LIN {X 0,Y 291.702,Z 865.941,A -85,B 0,C 180,E1 -16752.169,E2 -16752.169} C_VEL
LIN {X 0,Y 292.746,Z 856.676,A -85,B 0,C 180,E1 -16754.244,E2 -16754.244} C_VEL
LIN {X 0,Y 293.945,Z 846.153,A -85,B 0,C 180,E1 -16756.136,E2 -16756.136} C_VEL
LIN {X 0,Y 295.045,Z 835.726,A -85,B 0,C 180,E1 -16757.673,E2 -16757.673} C_VEL
LIN {X 0,Y 296.142,Z 824.245,A -85,B 0,C 180,E1 -16759.044,E2 -16759.044} C_VEL
LIN {X 0,Y 296.402,Z 819.576,A -85,B 0,C 180,E1 -16759.528,E2 -16759.528} C_VEL
LIN {X 0,Y 293.776,Z 806.153,A -85,B 0,C 180,E1 -16760.832,E2 -16760.832} C_VEL
LIN {X 0,Y 290.876,Z 792.284,A -85,B 0,C 180,E1 -16761.882,E2 -16761.882} C_VEL
LIN {X 0,Y 290.051,Z 788.06,A -85,B 0,C 180,E1 -16762.151,E2 -16762.151} C_VEL
LIN {X 0,Y 290.084,Z 786.203,A -85,B 0,C 180,E1 -16764.32,E2 -16764.32} C_VEL
LIN {X 0,Y 290.234,Z 785.335,A -85,B 0,C 180,E1 -16765.839,E2 -16765.839} C_VEL
LIN {X 0,Y 290.606,Z 785.282,A -85,B 0,C 180,E1 -16769.469,E2 -16769.469} C_VEL
LIN {X 0,Y 290.945,Z 785.244,A -85,B 0,C 180,E1 -16772.279,E2 -16772.279} C_VEL
LIN {X 0,Y 291.204,Z 785.208,A -85,B 0,C 180,E1 -16775.394,E2 -16775.394} C_VEL
LIN {X 0,Y 291.336,Z 785.194,A -85,B 0,C 180,E1 -16778.842,E2 -16778.842} C_VEL
LIN {X 0,Y 291.315,Z 785.197,A -85,B 0,C 180,E1 -16782.491,E2 -16782.491} C_VEL
LIN {X 0,Y 291.303,Z 785.198,A -85,B 0,C 180,E1 -16786.365,E2 -16786.365} C_VEL
LIN {X 0,Y 291.372,Z 785.188,A -85,B 0,C 180,E1 -16790.518,E2 -16790.518} C_VEL
LIN {X 0,Y 291.398,Z 785.189,A -85,B 0,C 180,E1 -16792.918,E2 -16792.918} C_VEL
LIN {X 0,Y 291.337,Z 785.192,A -85,B 0,C 180,E1 -16796.3,E2 -16796.3} C_VEL
LIN {X 0,Y 291.358,Z 785.188,A -85,B 0,C 180,E1 -16800.267,E2 -16800.267} C_VEL
LIN {X 0,Y 291.351,Z 785.19,A -85,B 0,C 180,E1 -16804.266,E2 -16804.266} C_VEL
LIN {X 0,Y 291.361,Z 785.193,A -85,B 0,C 180,E1 -16807.298,E2 -16807.298} C_VEL
LIN {X 0,Y 291.398,Z 785.184,A -85,B 0,C 180,E1 -16810.266,E2 -16810.266} C_VEL
LIN {X 0,Y 291.489,Z 785.172,A -85,B 0,C 180,E1 -16814.665,E2 -16814.665} C_VEL
LIN {X 0,Y 291.52,Z 785.169,A -85,B 0,C 180,E1 -16818.88,E2 -16818.88} C_VEL
LIN {X 0,Y 291.642,Z 785.158,A -85,B 0,C 180,E1 -16821.687,E2 -16821.687} C_VEL
LIN {X 0,Y 291.586,Z 785.16,A -85,B 0,C 180,E1 -16824.467,E2 -16824.467} C_VEL
LIN {X 0,Y 291.86,Z 785.127,A -85,B 0,C 180,E1 -16828.62,E2 -16828.62} C_VEL
LIN {X 0,Y 291.859,Z 785.127,A -85,B 0,C 180,E1 -16831.38,E2 -16831.38} C_VEL
LIN {X 0,Y 291.676,Z 785.15,A -85,B 0,C 180,E1 -16836.92,E2 -16836.92} C_VEL
LIN {X 0,Y 291.558,Z 785.165,A -85,B 0,C 180,E1 -16839.714,E2 -16839.714} C_VEL
LIN {X 0,Y 291.506,Z 785.171,A -85,B 0,C 180,E1 -16843.951,E2 -16843.951} C_VEL
LIN {X 0,Y 291.42,Z 785.184,A -85,B 0,C 180,E1 -16846.822,E2 -16846.822} C_VEL
LIN {X 0,Y 291.416,Z 785.182,A -85,B 0,C 180,E1 -16849.861,E2 -16849.861} C_VEL
LIN {X 0,Y 291.352,Z 785.191,A -85,B 0,C 180,E1 -16854.21,E2 -16854.21} C_VEL
LIN {X 0,Y 291.346,Z 785.192,A -85,B 0,C 180,E1 -16857.279,E2 -16857.279} C_VEL
LIN {X 0,Y 291.311,Z 785.196,A -85,B 0,C 180,E1 -16860.44,E2 -16860.44} C_VEL
LIN {X 0,Y 291.337,Z 785.192,A -85,B 0,C 180,E1 -16863.7,E2 -16863.7} C_VEL
LIN {X 0,Y 291.366,Z 785.191,A -85,B 0,C 180,E1 -16867.254,E2 -16867.254} C_VEL
LIN {X 0,Y 291.327,Z 785.193,A -85,B 0,C 180,E1 -16870.644,E2 -16870.644} C_VEL
LIN {X 0,Y 291.284,Z 785.198,A -85,B 0,C 180,E1 -16874.403,E2 -16874.403} C_VEL
LIN {X 0,Y 291.321,Z 785.193,A -85,B 0,C 180,E1 -16878.406,E2 -16878.406} C_VEL
LIN {X 0,Y 291.337,Z 785.194,A -85,B 0,C 180,E1 -16881.158,E2 -16881.158} C_VEL
LIN {X 0,Y 291.364,Z 785.189,A -85,B 0,C 180,E1 -16882.915,E2 -16882.915} C_VEL
LIN {X 0,Y 291.12,Z 785.219,A -85,B 0,C 180,E1 -16886.274,E2 -16886.274} C_VEL
LIN {X 0,Y 290.791,Z 785.263,A -85,B 0,C 180,E1 -16889.502,E2 -16889.502} C_VEL
LIN {X 0,Y 290.405,Z 785.308,A -85,B 0,C 180,E1 -16892.627,E2 -16892.627} C_VEL
LIN {X 0,Y 289.99,Z 785.385,A -85,B 0,C 180,E1 -16896.052,E2 -16896.052} C_VEL
LIN {X 0,Y 290.009,Z 787.302,A -85,B 0,C 180,E1 -16898.005,E2 -16898.005} C_VEL
LIN {X 0,Y 292.931,Z 801.867,A -85,B 0,C 180,E1 -16899.012,E2 -16899.012} C_VEL
LIN {X 0,Y 295.424,Z 814.684,A -85,B 0,C 180,E1 -16900.163,E2 -16900.163} C_VEL
LIN {X 0,Y 296.257,Z 818.937,A -85,B 0,C 180,E1 -16900.604,E2 -16900.604} C_VEL
LIN {X 0,Y 295.466,Z 830.012,A -85,B 0,C 180,E1 -16901.81,E2 -16901.81} C_VEL
LIN {X 0,Y 294.374,Z 841.527,A -85,B 0,C 180,E1 -16903.354,E2 -16903.354} C_VEL
LIN {X 0,Y 293.182,Z 851.897,A -85,B 0,C 180,E1 -16905.068,E2 -16905.068} C_VEL
LIN {X 0,Y 292.179,Z 860.521,A -85,B 0,C 180,E1 -16906.792,E2 -16906.792} C_VEL
LIN {X 0,Y 291.27,Z 869.021,A -85,B 0,C 180,E1 -16908.872,E2 -16908.872} C_VEL
LIN {X 0,Y 290.529,Z 875.88,A -85,B 0,C 180,E1 -16910.955,E2 -16910.955} C_VEL
LIN {X 0,Y 290.145,Z 881.419,A -85,B 0,C 180,E1 -16913.045,E2 -16913.045} C_VEL
LIN {X 0,Y 289.874,Z 885.775,A -85,B 0,C 180,E1 -16915.134,E2 -16915.134} C_VEL
LIN {X 0,Y 289.725,Z 889.058,A -85,B 0,C 180,E1 -16917.221,E2 -16917.221} C_VEL
LIN {X 0,Y 289.68,Z 890.166,A -85,B 0,C 180,E1 -16918.16,E2 -16918.16} C_VEL
LIN {X 0,Y 289.052,Z 891.419,A -85,B 0,C 180,E1 -16919.297,E2 -16919.297} C_VEL
LIN {X 0,Y 286.375,Z 892.977,A -85,B 0,C 180,E1 -16921.173,E2 -16921.173} C_VEL
LIN {X 0,Y 284.14,Z 893.629,A -85,B 0,C 180,E1 -16922.707,E2 -16922.707} C_VEL
LIN {X 0,Y 283.223,Z 893.7,A -85,B 0,C 180,E1 -16923.895,E2 -16923.895} C_VEL
LIN {X 0,Y 283.171,Z 893.633,A -85,B 0,C 180,E1 -16924.296,E2 -16924.296} C_VEL
LIN {X 0,Y 283.733,Z 892.595,A -85,B 0,C 180,E1 -16927.116,E2 -16927.116} C_VEL
LIN {X 0,Y 284.867,Z 890.681,A -85,B 0,C 180,E1 -16929.301,E2 -16929.301} C_VEL
LIN {X 0,Y 286.349,Z 886.93,A -85,B 0,C 180,E1 -16932.043,E2 -16932.043} C_VEL
LIN {X 0,Y 288.523,Z 881.299,A -85,B 0,C 180,E1 -16934.82,E2 -16934.82} C_VEL
LIN {X 0,Y 290.974,Z 874.766,A -85,B 0,C 180,E1 -16937.212,E2 -16937.212} C_VEL
LIN {X 0,Y 293.868,Z 866.526,A -85,B 0,C 180,E1 -16939.563,E2 -16939.563} C_VEL
LIN {X 0,Y 296.798,Z 857.782,A -85,B 0,C 180,E1 -16941.534,E2 -16941.534} C_VEL
LIN {X 0,Y 300.013,Z 847.159,A -85,B 0,C 180,E1 -16943.469,E2 -16943.469} C_VEL
LIN {X 0,Y 302.761,Z 837.452,A -85,B 0,C 180,E1 -16944.894,E2 -16944.894} C_VEL
LIN {X 0,Y 301.396,Z 829.053,A -85,B 0,C 180,E1 -16946.69,E2 -16946.69} C_VEL
LIN {X 0,Y 299.193,Z 821.542,A -85,B 0,C 180,E1 -16948.479,E2 -16948.479} C_VEL
LIN {X 0,Y 296.103,Z 814.055,A -85,B 0,C 180,E1 -16950.547,E2 -16950.547} C_VEL
LIN {X 0,Y 292.669,Z 807.234,A -85,B 0,C 180,E1 -16952.81,E2 -16952.81} C_VEL
LIN {X 0,Y 290.172,Z 802.954,A -85,B 0,C 180,E1 -16954.564,E2 -16954.564} C_VEL
LIN {X 0,Y 287.786,Z 800.116,A -85,B 0,C 180,E1 -16956.303,E2 -16956.303} C_VEL
LIN {X 0,Y 287.055,Z 798.413,A -85,B 0,C 180,E1 -16957.188,E2 -16957.188} C_VEL
LIN {X 0,Y 287.219,Z 798.097,A -85,B 0,C 180,E1 -16960.664,E2 -16960.664} C_VEL
LIN {X 0,Y 287.395,Z 798.308,A -85,B 0,C 180,E1 -16963.215,E2 -16963.215} C_VEL
LIN {X 0,Y 287.484,Z 798.802,A -85,B 0,C 180,E1 -16965.151,E2 -16965.151} C_VEL
LIN {X 0,Y 287.572,Z 799.696,A -85,B 0,C 180,E1 -16967.155,E2 -16967.155} C_VEL
LIN {X 0,Y 287.764,Z 802.16,A -85,B 0,C 180,E1 -16970.58,E2 -16970.58} C_VEL
LIN {X 0,Y 287.97,Z 805.028,A -85,B 0,C 180,E1 -16973.185,E2 -16973.185} C_VEL
LIN {X 0,Y 290.424,Z 811.895,A -85,B 0,C 180,E1 -16975.365,E2 -16975.365} C_VEL
LIN {X 0,Y 292.114,Z 817.637,A -85,B 0,C 180,E1 -16976.764,E2 -16976.764} C_VEL
LIN {X 0,Y 293.714,Z 824.775,A -85,B 0,C 180,E1 -16978.236,E2 -16978.236} C_VEL
LIN {X 0,Y 295.55,Z 834.314,A -85,B 0,C 180,E1 -16980.042,E2 -16980.042} C_VEL
LIN {X 0,Y 296.936,Z 846.854,A -85,B 0,C 180,E1 -16982.195,E2 -16982.195} C_VEL
LIN {X 0,Y 297.261,Z 857.519,A -85,B 0,C 180,E1 -16983.953,E2 -16983.953} C_VEL
LIN {X 0,Y 296.48,Z 867.317,A -85,B 0,C 180,E1 -16985.542,E2 -16985.542} C_VEL
LIN {X 0,Y 295.029,Z 876.946,A -85,B 0,C 180,E1 -16987.226,E2 -16987.226} C_VEL
LIN {X 0,Y 291.992,Z 887.534,A -85,B 0,C 180,E1 -16989.205,E2 -16989.205} C_VEL
LIN {X 0,Y 289.317,Z 896.401,A -85,B 0,C 180,E1 -16991.261,E2 -16991.261} C_VEL
LIN {X 0,Y 287.218,Z 903.602,A -85,B 0,C 180,E1 -16993.291,E2 -16993.291} C_VEL
LIN {X 0,Y 285.274,Z 910.592,A -85,B 0,C 180,E1 -16995.738,E2 -16995.738} C_VEL
LIN {X 0,Y 284.001,Z 915.383,A -85,B 0,C 180,E1 -16997.857,E2 -16997.857} C_VEL
LIN {X 0,Y 283.201,Z 919.135,A -85,B 0,C 180,E1 -16999.996,E2 -16999.996} C_VEL
LIN {X 0,Y 282.607,Z 922.647,A -85,B 0,C 180,E1 -17002.857,E2 -17002.857} C_VEL
LIN {X 0,Y 282.567,Z 923.809,A -85,B 0,C 180,E1 -17004.29,E2 -17004.29} C_VEL
LIN {X 0,Y 282.529,Z 924.564,A -85,B 0,C 180,E1 -17005.72,E2 -17005.72} C_VEL
LIN {X 0,Y 282.847,Z 924.892,A -85,B 0,C 180,E1 -17008.576,E2 -17008.576} C_VEL
LIN {X 0,Y 282.886,Z 925.833,A -85,B 0,C 180,E1 -17010,E2 -17010} C_VEL
LIN {X 0,Y 282.634,Z 926.326,A -85,B 0,C 180,E1 -17011.425,E2 -17011.425} C_VEL
LIN {X 0,Y 282.506,Z 926.418,A -85,B 0,C 180,E1 -17012.852,E2 -17012.852} C_VEL
LIN {X 0,Y 282.491,Z 926.109,A -85,B 0,C 180,E1 -17014.28,E2 -17014.28} C_VEL
LIN {X 0,Y 282.487,Z 925.361,A -85,B 0,C 180,E1 -17015.711,E2 -17015.711} C_VEL
LIN {X 0,Y 282.82,Z 922.66,A -85,B 0,C 180,E1 -17018.575,E2 -17018.575} C_VEL
LIN {X 0,Y 283.413,Z 919.571,A -85,B 0,C 180,E1 -17020.719,E2 -17020.719} C_VEL
LIN {X 0,Y 284.314,Z 915.533,A -85,B 0,C 180,E1 -17022.854,E2 -17022.854} C_VEL
LIN {X 0,Y 285.869,Z 910.437,A -85,B 0,C 180,E1 -17024.96,E2 -17024.96} C_VEL
LIN {X 0,Y 287.926,Z 903.011,A -85,B 0,C 180,E1 -17027.445,E2 -17027.445} C_VEL
LIN {X 0,Y 290.527,Z 894.081,A -85,B 0,C 180,E1 -17029.796,E2 -17029.796} C_VEL
LIN {X 0,Y 293.508,Z 884.684,A -85,B 0,C 180,E1 -17031.786,E2 -17031.786} C_VEL
LIN {X 0,Y 295.658,Z 877.383,A -85,B 0,C 180,E1 -17033.093,E2 -17033.093} C_VEL
LIN {X 0,Y 297.65,Z 865.19,A -85,B 0,C 180,E1 -17035.151,E2 -17035.151} C_VEL
LIN {X 0,Y 297.917,Z 856.285,A -85,B 0,C 180,E1 -17036.63,E2 -17036.63} C_VEL
LIN {X 0,Y 297.073,Z 845.544,A -85,B 0,C 180,E1 -17038.505,E2 -17038.505} C_VEL
LIN {X 0,Y 295.39,Z 836.08,A -85,B 0,C 180,E1 -17040.302,E2 -17040.302} C_VEL
LIN {X 0,Y 294.81,Z 833.066,A -85,B 0,C 180,E1 -17040.882,E2 -17040.882} C_VEL
LIN {X 0,Y 292.262,Z 823.462,A -85,B 0,C 180,E1 -17043.018,E2 -17043.018} C_VEL
LIN {X 0,Y 290.605,Z 818.78,A -85,B 0,C 180,E1 -17044.283,E2 -17044.283} C_VEL
LIN {X 0,Y 290.319,Z 817.311,A -85,B 0,C 180,E1 -17044.605,E2 -17044.605} C_VEL
LIN {X 0,Y 288.762,Z 814.222,A -85,B 0,C 180,E1 -17045.741,E2 -17045.741} C_VEL
LIN {X 0,Y 287.814,Z 810.336,A -85,B 0,C 180,E1 -17046.863,E2 -17046.863} C_VEL
LIN {X 0,Y 287.991,Z 808.098,A -85,B 0,C 180,E1 -17049.383,E2 -17049.383} C_VEL
LIN {X 0,Y 287.921,Z 806.691,A -85,B 0,C 180,E1 -17051.228,E2 -17051.228} C_VEL
LIN {X 0,Y 287.538,Z 804.324,A -85,B 0,C 180,E1 -17055.139,E2 -17055.139} C_VEL
LIN {X 0,Y 287.216,Z 802.831,A -85,B 0,C 180,E1 -17058.647,E2 -17058.647} C_VEL
LIN {X 0,Y 286.958,Z 801.877,A -85,B 0,C 180,E1 -17062.244,E2 -17062.244} C_VEL
LIN {X 0,Y 286.873,Z 801.861,A -85,B 0,C 180,E1 -17062.894,E2 -17062.894} C_VEL
LIN {X 0,Y 288.086,Z 804.443,A -85,B 0,C 180,E1 -17064.161,E2 -17064.161} C_VEL
LIN {X 0,Y 290.015,Z 806.131,A -85,B 0,C 180,E1 -17065.48,E2 -17065.48} C_VEL
LIN {X 0,Y 291.774,Z 809.381,A -85,B 0,C 180,E1 -17066.847,E2 -17066.847} C_VEL
LIN {X 0,Y 293.171,Z 811.449,A -85,B 0,C 180,E1 -17067.744,E2 -17067.744} C_VEL
LIN {X 0,Y 296.861,Z 818.609,A -85,B 0,C 180,E1 -17070.186,E2 -17070.186} C_VEL
LIN {X 0,Y 299.558,Z 825.112,A -85,B 0,C 180,E1 -17072.015,E2 -17072.015} C_VEL
LIN {X 0,Y 301.666,Z 832.042,A -85,B 0,C 180,E1 -17073.726,E2 -17073.726} C_VEL
LIN {X 0,Y 302.857,Z 838.726,A -85,B 0,C 180,E1 -17075.209,E2 -17075.209} C_VEL
LIN {X 0,Y 299.74,Z 849.593,A -85,B 0,C 180,E1 -17076.874,E2 -17076.874} C_VEL
LIN {X 0,Y 296.516,Z 859.861,A -85,B 0,C 180,E1 -17078.809,E2 -17078.809} C_VEL
LIN {X 0,Y 293.544,Z 868.287,A -85,B 0,C 180,E1 -17080.778,E2 -17080.778} C_VEL
LIN {X 0,Y 290.768,Z 876.232,A -85,B 0,C 180,E1 -17083.138,E2 -17083.138} C_VEL
LIN {X 0,Y 288.675,Z 881.708,A -85,B 0,C 180,E1 -17085.188,E2 -17085.188} C_VEL
LIN {X 0,Y 286.452,Z 887.341,A -85,B 0,C 180,E1 -17087.962,E2 -17087.962} C_VEL
LIN {X 0,Y 285.068,Z 890.835,A -85,B 0,C 180,E1 -17090.455,E2 -17090.455} C_VEL
LIN {X 0,Y 283.754,Z 893.037,A -85,B 0,C 180,E1 -17092.885,E2 -17092.885} C_VEL
LIN {X 0,Y 283.297,Z 894.093,A -85,B 0,C 180,E1 -17095.73,E2 -17095.73} C_VEL
LIN {X 0,Y 283.018,Z 894.026,A -85,B 0,C 180,E1 -17097.152,E2 -17097.152} C_VEL
LIN {X 0,Y 282.678,Z 892.699,A -85,B 0,C 180,E1 -17099.999,E2 -17099.999} C_VEL
LIN {X 0,Y 282.632,Z 891.447,A -85,B 0,C 180,E1 -17101.423,E2 -17101.423} C_VEL
LIN {X 0,Y 282.713,Z 888.747,A -85,B 0,C 180,E1 -17103.562,E2 -17103.562} C_VEL
LIN {X 0,Y 282.878,Z 884.509,A -85,B 0,C 180,E1 -17105.958,E2 -17105.958} C_VEL
LIN {X 0,Y 283.343,Z 878.316,A -85,B 0,C 180,E1 -17108.557,E2 -17108.557} C_VEL
LIN {X 0,Y 284.019,Z 871.834,A -85,B 0,C 180,E1 -17110.694,E2 -17110.694} C_VEL
LIN {X 0,Y 284.851,Z 863.81,A -85,B 0,C 180,E1 -17112.828,E2 -17112.828} C_VEL
LIN {X 0,Y 286.036,Z 853.966,A -85,B 0,C 180,E1 -17114.949,E2 -17114.949} C_VEL
LIN {X 0,Y 287.276,Z 843.933,A -85,B 0,C 180,E1 -17116.704,E2 -17116.704} C_VEL
LIN {X 0,Y 288.387,Z 832.589,A -85,B 0,C 180,E1 -17118.322,E2 -17118.322} C_VEL
LIN {X 0,Y 289.426,Z 820.702,A -85,B 0,C 180,E1 -17119.688,E2 -17119.688} C_VEL
LIN {X 0,Y 286.786,Z 807.171,A -85,B 0,C 180,E1 -17121.051,E2 -17121.051} C_VEL
LIN {X 0,Y 284.073,Z 794.034,A -85,B 0,C 180,E1 -17122.087,E2 -17122.087} C_VEL
LIN {X 0,Y 283.006,Z 788.468,A -85,B 0,C 180,E1 -17122.444,E2 -17122.444} C_VEL
LIN {X 0,Y 283.05,Z 786.328,A -85,B 0,C 180,E1 -17124.966,E2 -17124.966} C_VEL
LIN {X 0,Y 283.394,Z 786.186,A -85,B 0,C 180,E1 -17128.11,E2 -17128.11} C_VEL
LIN {X 0,Y 283.749,Z 786.135,A -85,B 0,C 180,E1 -17131.339,E2 -17131.339} C_VEL
LIN {X 0,Y 284.159,Z 786.086,A -85,B 0,C 180,E1 -17135.296,E2 -17135.296} C_VEL
LIN {X 0,Y 284.268,Z 786.074,A -85,B 0,C 180,E1 -17138.174,E2 -17138.174} C_VEL
LIN {X 0,Y 284.267,Z 786.072,A -85,B 0,C 180,E1 -17141.874,E2 -17141.874} C_VEL
LIN {X 0,Y 284.249,Z 786.075,A -85,B 0,C 180,E1 -17146.188,E2 -17146.188} C_VEL
LIN {X 0,Y 284.3,Z 786.067,A -85,B 0,C 180,E1 -17150.023,E2 -17150.023} C_VEL
LIN {X 0,Y 284.324,Z 786.066,A -85,B 0,C 180,E1 -17153.613,E2 -17153.613} C_VEL
LIN {X 0,Y 284.299,Z 786.072,A -85,B 0,C 180,E1 -17157.189,E2 -17157.189} C_VEL
LIN {X 0,Y 284.33,Z 786.064,A -85,B 0,C 180,E1 -17160.373,E2 -17160.373} C_VEL
LIN {X 0,Y 284.298,Z 786.071,A -85,B 0,C 180,E1 -17163.578,E2 -17163.578} C_VEL
LIN {X 0,Y 284.321,Z 786.065,A -85,B 0,C 180,E1 -17166.703,E2 -17166.703} C_VEL
LIN {X 0,Y 284.368,Z 786.061,A -85,B 0,C 180,E1 -17169.904,E2 -17169.904} C_VEL
LIN {X 0,Y 284.438,Z 786.051,A -85,B 0,C 180,E1 -17174.492,E2 -17174.492} C_VEL
LIN {X 0,Y 284.473,Z 786.046,A -85,B 0,C 180,E1 -17178.601,E2 -17178.601} C_VEL
LIN {X 0,Y 284.599,Z 786.034,A -85,B 0,C 180,E1 -17181.479,E2 -17181.479} C_VEL
LIN {X 0,Y 284.556,Z 786.037,A -85,B 0,C 180,E1 -17184.33,E2 -17184.33} C_VEL
LIN {X 0,Y 284.827,Z 786.003,A -85,B 0,C 180,E1 -17188.586,E2 -17188.586} C_VEL
LIN {X 0,Y 284.826,Z 786.003,A -85,B 0,C 180,E1 -17191.414,E2 -17191.414} C_VEL
LIN {X 0,Y 284.631,Z 786.027,A -85,B 0,C 180,E1 -17197.092,E2 -17197.092} C_VEL
LIN {X 0,Y 284.504,Z 786.045,A -85,B 0,C 180,E1 -17199.958,E2 -17199.958} C_VEL
LIN {X 0,Y 284.454,Z 786.052,A -85,B 0,C 180,E1 -17204.304,E2 -17204.304} C_VEL
LIN {X 0,Y 284.332,Z 786.067,A -85,B 0,C 180,E1 -17208.743,E2 -17208.743} C_VEL
LIN {X 0,Y 284.303,Z 786.067,A -85,B 0,C 180,E1 -17211.765,E2 -17211.765} C_VEL
LIN {X 0,Y 284.298,Z 786.072,A -85,B 0,C 180,E1 -17214.85,E2 -17214.85} C_VEL
LIN {X 0,Y 284.276,Z 786.071,A -85,B 0,C 180,E1 -17218.017,E2 -17218.017} C_VEL
LIN {X 0,Y 284.278,Z 786.072,A -85,B 0,C 180,E1 -17221.277,E2 -17221.277} C_VEL
LIN {X 0,Y 284.334,Z 786.066,A -85,B 0,C 180,E1 -17225.349,E2 -17225.349} C_VEL
LIN {X 0,Y 284.302,Z 786.068,A -85,B 0,C 180,E1 -17228.171,E2 -17228.171} C_VEL
LIN {X 0,Y 284.263,Z 786.072,A -85,B 0,C 180,E1 -17232.126,E2 -17232.126} C_VEL
LIN {X 0,Y 284.25,Z 786.074,A -85,B 0,C 180,E1 -17236.191,E2 -17236.191} C_VEL
LIN {X 0,Y 284.302,Z 786.068,A -85,B 0,C 180,E1 -17240.026,E2 -17240.026} C_VEL
LIN {X 0,Y 284.244,Z 786.08,A -85,B 0,C 180,E1 -17243.603,E2 -17243.603} C_VEL
LIN {X 0,Y 283.989,Z 786.109,A -85,B 0,C 180,E1 -17247.29,E2 -17247.29} C_VEL
LIN {X 0,Y 283.669,Z 786.147,A -85,B 0,C 180,E1 -17250.299,E2 -17250.299} C_VEL
LIN {X 0,Y 283.265,Z 786.2,A -85,B 0,C 180,E1 -17253.477,E2 -17253.477} C_VEL
LIN {X 0,Y 282.936,Z 786.382,A -85,B 0,C 180,E1 -17256.39,E2 -17256.39} C_VEL
LIN {X 0,Y 282.948,Z 787.872,A -85,B 0,C 180,E1 -17257.729,E2 -17257.729} C_VEL
LIN {X 0,Y 285.822,Z 802.312,A -85,B 0,C 180,E1 -17258.742,E2 -17258.742} C_VEL
LIN {X 0,Y 288.328,Z 815.122,A -85,B 0,C 180,E1 -17259.922,E2 -17259.922} C_VEL
LIN {X 0,Y 289.288,Z 820.39,A -85,B 0,C 180,E1 -17260.487,E2 -17260.487} C_VEL
LIN {X 0,Y 288.34,Z 831.842,A -85,B 0,C 180,E1 -17261.787,E2 -17261.787} C_VEL
LIN {X 0,Y 287.113,Z 843.637,A -85,B 0,C 180,E1 -17263.469,E2 -17263.469} C_VEL
LIN {X 0,Y 285.804,Z 854.596,A -85,B 0,C 180,E1 -17265.403,E2 -17265.403} C_VEL
LIN {X 0,Y 284.707,Z 864.273,A -85,B 0,C 180,E1 -17267.528,E2 -17267.528} C_VEL
LIN {X 0,Y 283.855,Z 872.143,A -85,B 0,C 180,E1 -17269.661,E2 -17269.661} C_VEL
LIN {X 0,Y 283.215,Z 879.438,A -85,B 0,C 180,E1 -17272.157,E2 -17272.157} C_VEL
LIN {X 0,Y 282.839,Z 884.347,A -85,B 0,C 180,E1 -17274.297,E2 -17274.297} C_VEL
LIN {X 0,Y 282.696,Z 888.133,A -85,B 0,C 180,E1 -17276.438,E2 -17276.438} C_VEL
LIN {X 0,Y 282.599,Z 890.878,A -85,B 0,C 180,E1 -17278.576,E2 -17278.576} C_VEL
LIN {X 0,Y 282.629,Z 892.175,A -85,B 0,C 180,E1 -17280.001,E2 -17280.001} C_VEL
LIN {X 0,Y 282.96,Z 893.537,A -85,B 0,C 180,E1 -17282.849,E2 -17282.849} C_VEL
LIN {X 0,Y 283.171,Z 893.633,A -85,B 0,C 180,E1 -17284.296,E2 -17284.296} C_VEL
LIN {X 0,Y 282.679,Z 893.458,A -85,B 0,C 180,E1 -17285.488,E2 -17285.488} C_VEL
LIN {X 0,Y 280.431,Z 892.807,A -85,B 0,C 180,E1 -17287.45,E2 -17287.45} C_VEL
LIN {X 0,Y 278.732,Z 891.925,A -85,B 0,C 180,E1 -17289.027,E2 -17289.027} C_VEL
LIN {X 0,Y 278.318,Z 890.871,A -85,B 0,C 180,E1 -17290.218,E2 -17290.218} C_VEL
LIN {X 0,Y 278.451,Z 890.393,A -85,B 0,C 180,E1 -17290.611,E2 -17290.611} C_VEL
LIN {X 0,Y 280.006,Z 886.909,A -85,B 0,C 180,E1 -17293.057,E2 -17293.057} C_VEL
LIN {X 0,Y 281.806,Z 882.732,A -85,B 0,C 180,E1 -17295.182,E2 -17295.182} C_VEL
LIN {X 0,Y 284.015,Z 877.472,A -85,B 0,C 180,E1 -17297.275,E2 -17297.275} C_VEL
LIN {X 0,Y 286.936,Z 869.907,A -85,B 0,C 180,E1 -17299.682,E2 -17299.682} C_VEL
LIN {X 0,Y 290.536,Z 860.297,A -85,B 0,C 180,E1 -17302.022,E2 -17302.022} C_VEL
LIN {X 0,Y 293.315,Z 852.081,A -85,B 0,C 180,E1 -17303.663,E2 -17303.663} C_VEL
LIN {X 0,Y 297.07,Z 839.913,A -85,B 0,C 180,E1 -17305.605,E2 -17305.605} C_VEL
LIN {X 0,Y 295.967,Z 832.182,A -85,B 0,C 180,E1 -17307.397,E2 -17307.397} C_VEL
LIN {X 0,Y 294.364,Z 826.026,A -85,B 0,C 180,E1 -17308.99,E2 -17308.99} C_VEL
LIN {X 0,Y 291.41,Z 818.131,A -85,B 0,C 180,E1 -17311.349,E2 -17311.349} C_VEL
LIN {X 0,Y 289.184,Z 813.256,A -85,B 0,C 180,E1 -17313.084,E2 -17313.084} C_VEL
LIN {X 0,Y 287.243,Z 809.619,A -85,B 0,C 180,E1 -17314.658,E2 -17314.658} C_VEL
LIN {X 0,Y 284.014,Z 804.72,A -85,B 0,C 180,E1 -17317.641,E2 -17317.641} C_VEL
LIN {X 0,Y 281.733,Z 802.604,A -85,B 0,C 180,E1 -17320.437,E2 -17320.437} C_VEL
LIN {X 0,Y 280.883,Z 801.093,A -85,B 0,C 180,E1 -17323.148,E2 -17323.148} C_VEL
LIN {X 0,Y 281.116,Z 802.523,A -85,B 0,C 180,E1 -17326.846,E2 -17326.846} C_VEL
LIN {X 0,Y 281.173,Z 803.067,A -85,B 0,C 180,E1 -17327.555,E2 -17327.555} C_VEL
LIN {X 0,Y 283.213,Z 808.036,A -85,B 0,C 180,E1 -17331.051,E2 -17331.051} C_VEL
LIN {X 0,Y 284.412,Z 810.164,A -85,B 0,C 180,E1 -17332.256,E2 -17332.256} C_VEL
LIN {X 0,Y 285.515,Z 813.347,A -85,B 0,C 180,E1 -17333.45,E2 -17333.45} C_VEL
LIN {X 0,Y 287.221,Z 818.649,A -85,B 0,C 180,E1 -17335.126,E2 -17335.126} C_VEL
LIN {X 0,Y 288.097,Z 822.214,A -85,B 0,C 180,E1 -17336.041,E2 -17336.041} C_VEL
LIN {X 0,Y 289.902,Z 832.451,A -85,B 0,C 180,E1 -17338.26,E2 -17338.26} C_VEL
LIN {X 0,Y 291.136,Z 843.347,A -85,B 0,C 180,E1 -17340.349,E2 -17340.349} C_VEL
LIN {X 0,Y 291.584,Z 855.35,A -85,B 0,C 180,E1 -17342.5,E2 -17342.5} C_VEL
LIN {X 0,Y 291.047,Z 865.259,A -85,B 0,C 180,E1 -17344.237,E2 -17344.237} C_VEL
LIN {X 0,Y 288.68,Z 878.809,A -85,B 0,C 180,E1 -17346.696,E2 -17346.696} C_VEL
LIN {X 0,Y 285.478,Z 888.796,A -85,B 0,C 180,E1 -17348.708,E2 -17348.708} C_VEL
LIN {X 0,Y 282.671,Z 897.379,A -85,B 0,C 180,E1 -17350.804,E2 -17350.804} C_VEL
LIN {X 0,Y 280.125,Z 905.283,A -85,B 0,C 180,E1 -17353.23,E2 -17353.23} C_VEL
LIN {X 0,Y 278.415,Z 910.935,A -85,B 0,C 180,E1 -17355.379,E2 -17355.379} C_VEL
LIN {X 0,Y 277.045,Z 915.502,A -85,B 0,C 180,E1 -17357.548,E2 -17357.548} C_VEL
LIN {X 0,Y 276.189,Z 919.099,A -85,B 0,C 180,E1 -17359.739,E2 -17359.739} C_VEL
LIN {X 0,Y 275.531,Z 922.433,A -85,B 0,C 180,E1 -17362.673,E2 -17362.673} C_VEL
LIN {X 0,Y 275.492,Z 923.548,A -85,B 0,C 180,E1 -17364.232,E2 -17364.232} C_VEL
LIN {X 0,Y 275.489,Z 924.365,A -85,B 0,C 180,E1 -17367.075,E2 -17367.075} C_VEL
LIN {X 0,Y 275.786,Z 924.211,A -85,B 0,C 180,E1 -17368.54,E2 -17368.54} C_VEL
LIN {X 0,Y 275.83,Z 925.179,A -85,B 0,C 180,E1 -17370,E2 -17370} C_VEL
LIN {X 0,Y 275.431,Z 925.9,A -85,B 0,C 180,E1 -17372.925,E2 -17372.925} C_VEL
LIN {X 0,Y 275.392,Z 925.176,A -85,B 0,C 180,E1 -17375.558,E2 -17375.558} C_VEL
LIN {X 0,Y 275.523,Z 923.974,A -85,B 0,C 180,E1 -17377.327,E2 -17377.327} C_VEL
LIN {X 0,Y 276.179,Z 920.665,A -85,B 0,C 180,E1 -17380.261,E2 -17380.261} C_VEL
LIN {X 0,Y 277.032,Z 917.1,A -85,B 0,C 180,E1 -17382.453,E2 -17382.453} C_VEL
LIN {X 0,Y 278.447,Z 912.585,A -85,B 0,C 180,E1 -17384.62,E2 -17384.62} C_VEL
LIN {X 0,Y 280.51,Z 905.989,A -85,B 0,C 180,E1 -17387.121,E2 -17387.121} C_VEL
LIN {X 0,Y 282.38,Z 900.06,A -85,B 0,C 180,E1 -17388.954,E2 -17388.954} C_VEL
LIN {X 0,Y 284.918,Z 892.333,A -85,B 0,C 180,E1 -17390.957,E2 -17390.957} C_VEL
LIN {X 0,Y 288.191,Z 882.745,A -85,B 0,C 180,E1 -17392.966,E2 -17392.966} C_VEL
LIN {X 0,Y 290.131,Z 875.514,A -85,B 0,C 180,E1 -17394.318,E2 -17394.318} C_VEL
LIN {X 0,Y 291.592,Z 867.572,A -85,B 0,C 180,E1 -17395.712,E2 -17395.712} C_VEL
LIN {X 0,Y 292.187,Z 859.278,A -85,B 0,C 180,E1 -17397.194,E2 -17397.194} C_VEL
LIN {X 0,Y 291.732,Z 848.938,A -85,B 0,C 180,E1 -17399.125,E2 -17399.125} C_VEL
LIN {X 0,Y 290.308,Z 838.853,A -85,B 0,C 180,E1 -17401.186,E2 -17401.186} C_VEL
LIN {X 0,Y 288.546,Z 830.885,A -85,B 0,C 180,E1 -17403.043,E2 -17403.043} C_VEL
LIN {X 0,Y 286.639,Z 822.943,A -85,B 0,C 180,E1 -17405.118,E2 -17405.118} C_VEL
LIN {X 0,Y 284.877,Z 818.122,A -85,B 0,C 180,E1 -17406.811,E2 -17406.811} C_VEL
LIN {X 0,Y 284.654,Z 816.669,A -85,B 0,C 180,E1 -17407.225,E2 -17407.225} C_VEL
LIN {X 0,Y 281.858,Z 810.987,A -85,B 0,C 180,E1 -17410.414,E2 -17410.414} C_VEL
LIN {X 0,Y 280.879,Z 807.287,A -85,B 0,C 180,E1 -17412.97,E2 -17412.97} C_VEL
LIN {X 0,Y 280.546,Z 805.527,A -85,B 0,C 180,E1 -17416.125,E2 -17416.125} C_VEL
LIN {X 0,Y 280.672,Z 805.678,A -85,B 0,C 180,E1 -17417.461,E2 -17417.461} C_VEL
LIN {X 0,Y 282.083,Z 807.298,A -85,B 0,C 180,E1 -17420.566,E2 -17420.566} C_VEL
LIN {X 0,Y 283.825,Z 808.235,A -85,B 0,C 180,E1 -17422.408,E2 -17422.408} C_VEL
LIN {X 0,Y 285.57,Z 811.217,A -85,B 0,C 180,E1 -17424.306,E2 -17424.306} C_VEL
LIN {X 0,Y 286.24,Z 811.851,A -85,B 0,C 180,E1 -17424.843,E2 -17424.843} C_VEL
LIN {X 0,Y 289.155,Z 816.685,A -85,B 0,C 180,E1 -17427.194,E2 -17427.194} C_VEL
LIN {X 0,Y 292.372,Z 823.479,A -85,B 0,C 180,E1 -17429.681,E2 -17429.681} C_VEL
LIN {X 0,Y 294.608,Z 829.492,A -85,B 0,C 180,E1 -17431.502,E2 -17431.502} C_VEL
LIN {X 0,Y 296.524,Z 836.949,A -85,B 0,C 180,E1 -17433.472,E2 -17433.472} C_VEL
LIN {X 0,Y 297.091,Z 841.673,A -85,B 0,C 180,E1 -17434.594,E2 -17434.594} C_VEL
LIN {X 0,Y 293.622,Z 852.625,A -85,B 0,C 180,E1 -17436.363,E2 -17436.363} C_VEL
LIN {X 0,Y 290.22,Z 862.317,A -85,B 0,C 180,E1 -17438.326,E2 -17438.326} C_VEL
LIN {X 0,Y 287.122,Z 870.395,A -85,B 0,C 180,E1 -17440.331,E2 -17440.331} C_VEL
LIN {X 0,Y 284.188,Z 877.937,A -85,B 0,C 180,E1 -17442.735,E2 -17442.735} C_VEL
LIN {X 0,Y 281.975,Z 883.17,A -85,B 0,C 180,E1 -17444.827,E2 -17444.827} C_VEL
LIN {X 0,Y 280.124,Z 887.346,A -85,B 0,C 180,E1 -17446.949,E2 -17446.949} C_VEL
LIN {X 0,Y 279.097,Z 889.589,A -85,B 0,C 180,E1 -17448.377,E2 -17448.377} C_VEL
LIN {X 0,Y 277.573,Z 892.771,A -85,B 0,C 180,E1 -17451.261,E2 -17451.261} C_VEL
LIN {X 0,Y 276.762,Z 893.817,A -85,B 0,C 180,E1 -17452.704,E2 -17452.704} C_VEL
LIN {X 0,Y 276.43,Z 894.437,A -85,B 0,C 180,E1 -17454.162,E2 -17454.162} C_VEL
LIN {X 0,Y 276.227,Z 894.639,A -85,B 0,C 180,E1 -17455.621,E2 -17455.621} C_VEL
LIN {X 0,Y 275.709,Z 893.92,A -85,B 0,C 180,E1 -17458.538,E2 -17458.538} C_VEL
LIN {X 0,Y 275.586,Z 892.977,A -85,B 0,C 180,E1 -17459.999,E2 -17459.999} C_VEL
LIN {X 0,Y 275.546,Z 891.59,A -85,B 0,C 180,E1 -17461.46,E2 -17461.46} C_VEL
LIN {X 0,Y 275.646,Z 888.744,A -85,B 0,C 180,E1 -17463.653,E2 -17463.653} C_VEL
LIN {X 0,Y 275.787,Z 884.884,A -85,B 0,C 180,E1 -17465.849,E2 -17465.849} C_VEL
LIN {X 0,Y 276.165,Z 879.912,A -85,B 0,C 180,E1 -17468.044,E2 -17468.044} C_VEL
LIN {X 0,Y 276.873,Z 872.501,A -85,B 0,C 180,E1 -17470.603,E2 -17470.603} C_VEL
LIN {X 0,Y 277.722,Z 864.529,A -85,B 0,C 180,E1 -17472.791,E2 -17472.791} C_VEL
LIN {X 0,Y 278.891,Z 854.72,A -85,B 0,C 180,E1 -17474.967,E2 -17474.967} C_VEL
LIN {X 0,Y 280.135,Z 844.769,A -85,B 0,C 180,E1 -17476.767,E2 -17476.767} C_VEL
LIN {X 0,Y 281.331,Z 833.067,A -85,B 0,C 180,E1 -17478.485,E2 -17478.485} C_VEL
LIN {X 0,Y 282.401,Z 821.881,A -85,B 0,C 180,E1 -17479.819,E2 -17479.819} C_VEL
LIN {X 0,Y 280.172,Z 810.092,A -85,B 0,C 180,E1 -17481.064,E2 -17481.064} C_VEL
LIN {X 0,Y 277.366,Z 796.146,A -85,B 0,C 180,E1 -17482.248,E2 -17482.248} C_VEL
LIN {X 0,Y 275.922,Z 788.841,A -85,B 0,C 180,E1 -17482.771,E2 -17482.771} C_VEL
LIN {X 0,Y 275.926,Z 787.766,A -85,B 0,C 180,E1 -17484.048,E2 -17484.048} C_VEL
LIN {X 0,Y 276.058,Z 787.101,A -85,B 0,C 180,E1 -17485.643,E2 -17485.643} C_VEL
LIN {X 0,Y 276.44,Z 787.048,A -85,B 0,C 180,E1 -17488.882,E2 -17488.882} C_VEL
LIN {X 0,Y 276.913,Z 786.988,A -85,B 0,C 180,E1 -17493.119,E2 -17493.119} C_VEL
LIN {X 0,Y 277.134,Z 786.961,A -85,B 0,C 180,E1 -17495.756,E2 -17495.756} C_VEL
LIN {X 0,Y 277.218,Z 786.95,A -85,B 0,C 180,E1 -17499.329,E2 -17499.329} C_VEL
LIN {X 0,Y 277.204,Z 786.953,A -85,B 0,C 180,E1 -17503.197,E2 -17503.197} C_VEL
LIN {X 0,Y 277.209,Z 786.952,A -85,B 0,C 180,E1 -17507.324,E2 -17507.324} C_VEL
LIN {X 0,Y 277.255,Z 786.946,A -85,B 0,C 180,E1 -17511.792,E2 -17511.792} C_VEL
LIN {X 0,Y 277.277,Z 786.944,A -85,B 0,C 180,E1 -17514.34,E2 -17514.34} C_VEL
LIN {X 0,Y 277.233,Z 786.947,A -85,B 0,C 180,E1 -17517.835,E2 -17517.835} C_VEL
LIN {X 0,Y 277.232,Z 786.954,A -85,B 0,C 180,E1 -17521.206,E2 -17521.206} C_VEL
LIN {X 0,Y 277.239,Z 786.948,A -85,B 0,C 180,E1 -17524.472,E2 -17524.472} C_VEL
LIN {X 0,Y 277.254,Z 786.948,A -85,B 0,C 180,E1 -17527.652,E2 -17527.652} C_VEL
LIN {X 0,Y 277.296,Z 786.941,A -85,B 0,C 180,E1 -17530.763,E2 -17530.763} C_VEL
LIN {X 0,Y 277.401,Z 786.93,A -85,B 0,C 180,E1 -17535.324,E2 -17535.324} C_VEL
LIN {X 0,Y 277.448,Z 786.927,A -85,B 0,C 180,E1 -17539.787,E2 -17539.787} C_VEL
LIN {X 0,Y 277.59,Z 786.904,A -85,B 0,C 180,E1 -17542.727,E2 -17542.727} C_VEL
LIN {X 0,Y 277.794,Z 786.88,A -85,B 0,C 180,E1 -17548.55,E2 -17548.55} C_VEL
LIN {X 0,Y 277.793,Z 786.88,A -85,B 0,C 180,E1 -17551.45,E2 -17551.45} C_VEL
LIN {X 0,Y 277.59,Z 786.904,A -85,B 0,C 180,E1 -17557.273,E2 -17557.273} C_VEL
LIN {X 0,Y 277.445,Z 786.927,A -85,B 0,C 180,E1 -17560.214,E2 -17560.214} C_VEL
LIN {X 0,Y 277.4,Z 786.93,A -85,B 0,C 180,E1 -17564.676,E2 -17564.676} C_VEL
LIN {X 0,Y 277.296,Z 786.941,A -85,B 0,C 180,E1 -17569.237,E2 -17569.237} C_VEL
LIN {X 0,Y 277.274,Z 786.943,A -85,B 0,C 180,E1 -17573.926,E2 -17573.926} C_VEL
LIN {X 0,Y 277.262,Z 786.945,A -85,B 0,C 180,E1 -17577.484,E2 -17577.484} C_VEL
LIN {X 0,Y 277.24,Z 786.949,A -85,B 0,C 180,E1 -17580.474,E2 -17580.474} C_VEL
LIN {X 0,Y 277.239,Z 786.947,A -85,B 0,C 180,E1 -17583.897,E2 -17583.897} C_VEL
LIN {X 0,Y 277.258,Z 786.947,A -85,B 0,C 180,E1 -17587.471,E2 -17587.471} C_VEL
LIN {X 0,Y 277.204,Z 786.956,A -85,B 0,C 180,E1 -17591.238,E2 -17591.238} C_VEL
LIN {X 0,Y 277.195,Z 786.958,A -85,B 0,C 180,E1 -17595.228,E2 -17595.228} C_VEL
LIN {X 0,Y 277.218,Z 786.953,A -85,B 0,C 180,E1 -17599.514,E2 -17599.514} C_VEL
LIN {X 0,Y 277.228,Z 786.949,A -85,B 0,C 180,E1 -17602.527,E2 -17602.527} C_VEL
LIN {X 0,Y 277.012,Z 786.977,A -85,B 0,C 180,E1 -17606.074,E2 -17606.074} C_VEL
LIN {X 0,Y 276.667,Z 787.023,A -85,B 0,C 180,E1 -17609.733,E2 -17609.733} C_VEL
LIN {X 0,Y 276.287,Z 787.067,A -85,B 0,C 180,E1 -17612.912,E2 -17612.912} C_VEL
LIN {X 0,Y 275.877,Z 787.15,A -85,B 0,C 180,E1 -17616.507,E2 -17616.507} C_VEL
LIN {X 0,Y 275.857,Z 788.04,A -85,B 0,C 180,E1 -17617.422,E2 -17617.422} C_VEL
LIN {X 0,Y 278.754,Z 802.912,A -85,B 0,C 180,E1 -17618.503,E2 -17618.503} C_VEL
LIN {X 0,Y 281.427,Z 816.719,A -85,B 0,C 180,E1 -17619.824,E2 -17619.824} C_VEL
LIN {X 0,Y 282.244,Z 821.541,A -85,B 0,C 180,E1 -17620.359,E2 -17620.359} C_VEL
LIN {X 0,Y 281.197,Z 833.281,A -85,B 0,C 180,E1 -17621.758,E2 -17621.758} C_VEL
LIN {X 0,Y 279.963,Z 844.448,A -85,B 0,C 180,E1 -17623.41,E2 -17623.41} C_VEL
LIN {X 0,Y 278.894,Z 853.522,A -85,B 0,C 180,E1 -17625.033,E2 -17625.033} C_VEL
LIN {X 0,Y 277.887,Z 861.998,A -85,B 0,C 180,E1 -17626.845,E2 -17626.845} C_VEL
LIN {X 0,Y 276.968,Z 870.352,A -85,B 0,C 180,E1 -17629.031,E2 -17629.031} C_VEL
LIN {X 0,Y 276.272,Z 877.166,A -85,B 0,C 180,E1 -17631.222,E2 -17631.222} C_VEL
LIN {X 0,Y 275.831,Z 882.967,A -85,B 0,C 180,E1 -17633.566,E2 -17633.566} C_VEL
LIN {X 0,Y 275.658,Z 886.929,A -85,B 0,C 180,E1 -17635.615,E2 -17635.615} C_VEL
LIN {X 0,Y 275.577,Z 889.178,A -85,B 0,C 180,E1 -17637.078,E2 -17637.078} C_VEL
LIN {X 0,Y 275.54,Z 892.417,A -85,B 0,C 180,E1 -17640.001,E2 -17640.001} C_VEL
LIN {X 0,Y 275.664,Z 893.401,A -85,B 0,C 180,E1 -17641.462,E2 -17641.462} C_VEL
LIN {X 0,Y 275.879,Z 893.967,A -85,B 0,C 180,E1 -17642.922,E2 -17642.922} C_VEL
LIN {X 0,Y 276.097,Z 894.153,A -85,B 0,C 180,E1 -17644.381,E2 -17644.381} C_VEL
LIN {X 0,Y 276.309,Z 893.971,A -85,B 0,C 180,E1 -17645.841,E2 -17645.841} C_VEL
LIN {X 0,Y 276.74,Z 893.354,A -85,B 0,C 180,E1 -17647.296,E2 -17647.296} C_VEL
LIN {X 0,Y 277.933,Z 891.599,A -85,B 0,C 180,E1 -17649.535,E2 -17649.535} C_VEL
LIN {X 0,Y 278.451,Z 890.393,A -85,B 0,C 180,E1 -17650.611,E2 -17650.611} C_VEL
LIN {X 0,Y 278.5,Z 889.039,A -85,B 0,C 180,E1 -17651.792,E2 -17651.792} C_VEL
LIN {X 0,Y 277.069,Z 886.606,A -85,B 0,C 180,E1 -17653.757,E2 -17653.757} C_VEL
LIN {X 0,Y 275.935,Z 883.689,A -85,B 0,C 180,E1 -17655.7,E2 -17655.7} C_VEL
LIN {X 0,Y 276.431,Z 881.39,A -85,B 0,C 180,E1 -17656.821,E2 -17656.821} C_VEL
LIN {X 0,Y 279.574,Z 874.192,A -85,B 0,C 180,E1 -17659.457,E2 -17659.457} C_VEL
LIN {X 0,Y 282.65,Z 867.012,A -85,B 0,C 180,E1 -17661.517,E2 -17661.517} C_VEL
LIN {X 0,Y 286.003,Z 858.274,A -85,B 0,C 180,E1 -17663.537,E2 -17663.537} C_VEL
LIN {X 0,Y 289.722,Z 847.967,A -85,B 0,C 180,E1 -17665.468,E2 -17665.468} C_VEL
LIN {X 0,Y 291.127,Z 843.853,A -85,B 0,C 180,E1 -17666.119,E2 -17666.119} C_VEL
LIN {X 0,Y 291.447,Z 842.038,A -85,B 0,C 180,E1 -17666.451,E2 -17666.451} C_VEL
LIN {X 0,Y 290.349,Z 833.992,A -85,B 0,C 180,E1 -17668.515,E2 -17668.515} C_VEL
LIN {X 0,Y 288.671,Z 827.755,A -85,B 0,C 180,E1 -17670.354,E2 -17670.354} C_VEL
LIN {X 0,Y 286.775,Z 822.364,A -85,B 0,C 180,E1 -17672.167,E2 -17672.167} C_VEL
LIN {X 0,Y 285.678,Z 819.548,A -85,B 0,C 180,E1 -17673.234,E2 -17673.234} C_VEL
LIN {X 0,Y 283.681,Z 815.339,A -85,B 0,C 180,E1 -17675.159,E2 -17675.159} C_VEL
LIN {X 0,Y 281.82,Z 812.365,A -85,B 0,C 180,E1 -17677.059,E2 -17677.059} C_VEL
LIN {X 0,Y 280.209,Z 810.346,A -85,B 0,C 180,E1 -17678.966,E2 -17678.966} C_VEL
LIN {X 0,Y 279.064,Z 808.96,A -85,B 0,C 180,E1 -17680.928,E2 -17680.928} C_VEL
LIN {X 0,Y 278.557,Z 807.804,A -85,B 0,C 180,E1 -17682.973,E2 -17682.973} C_VEL
LIN {X 0,Y 278.335,Z 808.267,A -85,B 0,C 180,E1 -17685.008,E2 -17685.008} C_VEL
LIN {X 0,Y 278.738,Z 809.38,A -85,B 0,C 180,E1 -17687.096,E2 -17687.096} C_VEL
LIN {X 0,Y 280.026,Z 813.459,A -85,B 0,C 180,E1 -17690.109,E2 -17690.109} C_VEL
LIN {X 0,Y 281.781,Z 817.386,A -85,B 0,C 180,E1 -17692.318,E2 -17692.318} C_VEL
LIN {X 0,Y 283.358,Z 823.226,A -85,B 0,C 180,E1 -17694.347,E2 -17694.347} C_VEL
LIN {X 0,Y 284.072,Z 826.799,A -85,B 0,C 180,E1 -17695.318,E2 -17695.318} C_VEL
LIN {X 0,Y 285.341,Z 837.351,A -85,B 0,C 180,E1 -17697.741,E2 -17697.741} C_VEL
LIN {X 0,Y 286.042,Z 848.747,A -85,B 0,C 180,E1 -17700.04,E2 -17700.04} C_VEL
LIN {X 0,Y 285.846,Z 860.396,A -85,B 0,C 180,E1 -17702.268,E2 -17702.268} C_VEL
LIN {X 0,Y 284.739,Z 869.724,A -85,B 0,C 180,E1 -17704.017,E2 -17704.017} C_VEL
LIN {X 0,Y 282.338,Z 880.604,A -85,B 0,C 180,E1 -17706.14,E2 -17706.14} C_VEL
LIN {X 0,Y 278.995,Z 890.192,A -85,B 0,C 180,E1 -17708.188,E2 -17708.188} C_VEL
LIN {X 0,Y 275.643,Z 899.384,A -85,B 0,C 180,E1 -17710.643,E2 -17710.643} C_VEL
LIN {X 0,Y 273.366,Z 905.93,A -85,B 0,C 180,E1 -17712.803,E2 -17712.803} C_VEL
LIN {X 0,Y 271.569,Z 911.307,A -85,B 0,C 180,E1 -17715.001,E2 -17715.001} C_VEL
LIN {X 0,Y 270.081,Z 915.686,A -85,B 0,C 180,E1 -17717.221,E2 -17717.221} C_VEL
LIN {X 0,Y 269.19,Z 919.073,A -85,B 0,C 180,E1 -17719.47,E2 -17719.47} C_VEL
LIN {X 0,Y 268.746,Z 920.851,A -85,B 0,C 180,E1 -17720.973,E2 -17720.973} C_VEL
LIN {X 0,Y 268.481,Z 922.203,A -85,B 0,C 180,E1 -17722.479,E2 -17722.479} C_VEL
LIN {X 0,Y 268.423,Z 923.271,A -85,B 0,C 180,E1 -17724.243,E2 -17724.243} C_VEL
LIN {X 0,Y 268.413,Z 923.865,A -85,B 0,C 180,E1 -17726.998,E2 -17726.998} C_VEL
LIN {X 0,Y 268.73,Z 923.649,A -85,B 0,C 180,E1 -17728.876,E2 -17728.876} C_VEL
LIN {X 0,Y 268.773,Z 924.449,A -85,B 0,C 180,E1 -17730,E2 -17730} C_VEL
LIN {X 0,Y 268.47,Z 925.129,A -85,B 0,C 180,E1 -17731.5,E2 -17731.5} C_VEL
LIN {X 0,Y 268.358,Z 925.383,A -85,B 0,C 180,E1 -17733.002,E2 -17733.002} C_VEL
LIN {X 0,Y 268.298,Z 924.91,A -85,B 0,C 180,E1 -17735.487,E2 -17735.487} C_VEL
LIN {X 0,Y 268.457,Z 923.714,A -85,B 0,C 180,E1 -17737.521,E2 -17737.521} C_VEL
LIN {X 0,Y 268.734,Z 922.379,A -85,B 0,C 180,E1 -17739.028,E2 -17739.028} C_VEL
LIN {X 0,Y 269.724,Z 918.469,A -85,B 0,C 180,E1 -17742.032,E2 -17742.032} C_VEL
LIN {X 0,Y 270.99,Z 914.479,A -85,B 0,C 180,E1 -17744.263,E2 -17744.263} C_VEL
LIN {X 0,Y 273.414,Z 907.615,A -85,B 0,C 180,E1 -17747.194,E2 -17747.194} C_VEL
LIN {X 0,Y 275.742,Z 900.97,A -85,B 0,C 180,E1 -17749.428,E2 -17749.428} C_VEL
LIN {X 0,Y 278.396,Z 893.523,A -85,B 0,C 180,E1 -17751.472,E2 -17751.472} C_VEL
LIN {X 0,Y 281.8,Z 884.417,A -85,B 0,C 180,E1 -17753.518,E2 -17753.518} C_VEL
LIN {X 0,Y 283.94,Z 877.49,A -85,B 0,C 180,E1 -17754.884,E2 -17754.884} C_VEL
LIN {X 0,Y 285.873,Z 868.277,A -85,B 0,C 180,E1 -17756.623,E2 -17756.623} C_VEL
LIN {X 0,Y 286.504,Z 859.438,A -85,B 0,C 180,E1 -17758.325,E2 -17758.325} C_VEL
LIN {X 0,Y 286.178,Z 849.568,A -85,B 0,C 180,E1 -17760.331,E2 -17760.331} C_VEL
LIN {X 0,Y 285.301,Z 841.733,A -85,B 0,C 180,E1 -17762.081,E2 -17762.081} C_VEL
LIN {X 0,Y 283.594,Z 832.587,A -85,B 0,C 180,E1 -17764.44,E2 -17764.44} C_VEL
LIN {X 0,Y 282.31,Z 827.112,A -85,B 0,C 180,E1 -17766.109,E2 -17766.109} C_VEL
LIN {X 0,Y 281.088,Z 822.068,A -85,B 0,C 180,E1 -17767.899,E2 -17767.899} C_VEL
LIN {X 0,Y 278.979,Z 817.031,A -85,B 0,C 180,E1 -17770.919,E2 -17770.919} C_VEL
LIN {X 0,Y 278.354,Z 814.117,A -85,B 0,C 180,E1 -17772.978,E2 -17772.978} C_VEL
LIN {X 0,Y 278.035,Z 812.637,A -85,B 0,C 180,E1 -17775.054,E2 -17775.054} C_VEL
LIN {X 0,Y 278.154,Z 812.277,A -85,B 0,C 180,E1 -17777.116,E2 -17777.116} C_VEL
LIN {X 0,Y 279.828,Z 814.123,A -85,B 0,C 180,E1 -17781.131,E2 -17781.131} C_VEL
LIN {X 0,Y 281.499,Z 816.173,A -85,B 0,C 180,E1 -17783.186,E2 -17783.186} C_VEL
LIN {X 0,Y 283.522,Z 819.246,A -85,B 0,C 180,E1 -17785.239,E2 -17785.239} C_VEL
LIN {X 0,Y 285.652,Z 823.341,A -85,B 0,C 180,E1 -17787.228,E2 -17787.228} C_VEL
LIN {X 0,Y 288.291,Z 829.746,A -85,B 0,C 180,E1 -17789.662,E2 -17789.662} C_VEL
LIN {X 0,Y 290.093,Z 835.604,A -85,B 0,C 180,E1 -17791.51,E2 -17791.51} C_VEL
LIN {X 0,Y 291.474,Z 842.941,A -85,B 0,C 180,E1 -17793.548,E2 -17793.548} C_VEL
LIN {X 0,Y 291.435,Z 844.548,A -85,B 0,C 180,E1 -17793.909,E2 -17793.909} C_VEL
LIN {X 0,Y 287.531,Z 855.604,A -85,B 0,C 180,E1 -17795.831,E2 -17795.831} C_VEL
LIN {X 0,Y 283.955,Z 864.842,A -85,B 0,C 180,E1 -17797.823,E2 -17797.823} C_VEL
LIN {X 0,Y 280.208,Z 873.632,A -85,B 0,C 180,E1 -17800.207,E2 -17800.207} C_VEL
LIN {X 0,Y 277.623,Z 879.712,A -85,B 0,C 180,E1 -17802.314,E2 -17802.314} C_VEL
LIN {X 0,Y 275.305,Z 884.672,A -85,B 0,C 180,E1 -17804.451,E2 -17804.451} C_VEL
LIN {X 0,Y 272.785,Z 889.69,A -85,B 0,C 180,E1 -17807.349,E2 -17807.349} C_VEL
LIN {X 0,Y 271.217,Z 892.766,A -85,B 0,C 180,E1 -17809.962,E2 -17809.962} C_VEL
LIN {X 0,Y 269.774,Z 894.578,A -85,B 0,C 180,E1 -17812.514,E2 -17812.514} C_VEL
LIN {X 0,Y 269.157,Z 895.171,A -85,B 0,C 180,E1 -17815.506,E2 -17815.506} C_VEL
LIN {X 0,Y 268.862,Z 894.913,A -85,B 0,C 180,E1 -17817.002,E2 -17817.002} C_VEL
LIN {X 0,Y 268.622,Z 894.267,A -85,B 0,C 180,E1 -17818.499,E2 -17818.499} C_VEL
LIN {X 0,Y 268.497,Z 893.188,A -85,B 0,C 180,E1 -17819.998,E2 -17819.998} C_VEL
LIN {X 0,Y 268.462,Z 891.714,A -85,B 0,C 180,E1 -17821.499,E2 -17821.499} C_VEL
LIN {X 0,Y 268.56,Z 888.705,A -85,B 0,C 180,E1 -17823.75,E2 -17823.75} C_VEL
LIN {X 0,Y 268.797,Z 883.642,A -85,B 0,C 180,E1 -17826.507,E2 -17826.507} C_VEL
LIN {X 0,Y 269.258,Z 877.518,A -85,B 0,C 180,E1 -17829.008,E2 -17829.008} C_VEL
LIN {X 0,Y 270.138,Z 869.367,A -85,B 0,C 180,E1 -17831.63,E2 -17831.63} C_VEL
LIN {X 0,Y 271.14,Z 860.597,A -85,B 0,C 180,E1 -17833.871,E2 -17833.871} C_VEL
LIN {X 0,Y 272.247,Z 851.735,A -85,B 0,C 180,E1 -17835.725,E2 -17835.725} C_VEL
LIN {X 0,Y 273.542,Z 841.053,A -85,B 0,C 180,E1 -17837.569,E2 -17837.569} C_VEL
LIN {X 0,Y 274.763,Z 828.961,A -85,B 0,C 180,E1 -17839.248,E2 -17839.248} C_VEL
LIN {X 0,Y 275.345,Z 822.92,A -85,B 0,C 180,E1 -17839.96,E2 -17839.96} C_VEL
LIN {X 0,Y 273.08,Z 810.672,A -85,B 0,C 180,E1 -17841.302,E2 -17841.302} C_VEL
LIN {X 0,Y 270.295,Z 796.593,A -85,B 0,C 180,E1 -17842.538,E2 -17842.538} C_VEL
LIN {X 0,Y 268.868,Z 789.237,A -85,B 0,C 180,E1 -17843.083,E2 -17843.083} C_VEL
LIN {X 0,Y 268.883,Z 787.996,A -85,B 0,C 180,E1 -17844.719,E2 -17844.719} C_VEL
LIN {X 0,Y 269.273,Z 787.944,A -85,B 0,C 180,E1 -17848.019,E2 -17848.019} C_VEL
LIN {X 0,Y 269.643,Z 787.892,A -85,B 0,C 180,E1 -17851.416,E2 -17851.416} C_VEL
LIN {X 0,Y 269.995,Z 787.852,A -85,B 0,C 180,E1 -17854.934,E2 -17854.934} C_VEL
LIN {X 0,Y 270.164,Z 787.832,A -85,B 0,C 180,E1 -17858.701,E2 -17858.701} C_VEL
LIN {X 0,Y 270.167,Z 787.832,A -85,B 0,C 180,E1 -17862.557,E2 -17862.557} C_VEL
LIN {X 0,Y 270.159,Z 787.835,A -85,B 0,C 180,E1 -17866.75,E2 -17866.75} C_VEL
LIN {X 0,Y 270.168,Z 787.828,A -85,B 0,C 180,E1 -17869.433,E2 -17869.433} C_VEL
LIN {X 0,Y 270.219,Z 787.823,A -85,B 0,C 180,E1 -17873.729,E2 -17873.729} C_VEL
LIN {X 0,Y 270.195,Z 787.829,A -85,B 0,C 180,E1 -17876.891,E2 -17876.891} C_VEL
LIN {X 0,Y 270.176,Z 787.827,A -85,B 0,C 180,E1 -17880.38,E2 -17880.38} C_VEL
LIN {X 0,Y 270.195,Z 787.827,A -85,B 0,C 180,E1 -17883.757,E2 -17883.757} C_VEL
LIN {X 0,Y 270.193,Z 787.827,A -85,B 0,C 180,E1 -17887.035,E2 -17887.035} C_VEL
LIN {X 0,Y 270.243,Z 787.819,A -85,B 0,C 180,E1 -17890.24,E2 -17890.24} C_VEL
LIN {X 0,Y 270.36,Z 787.805,A -85,B 0,C 180,E1 -17894.933,E2 -17894.933} C_VEL
LIN {X 0,Y 270.401,Z 787.803,A -85,B 0,C 180,E1 -17899.517,E2 -17899.517} C_VEL
LIN {X 0,Y 270.552,Z 787.781,A -85,B 0,C 180,E1 -17902.537,E2 -17902.537} C_VEL
LIN {X 0,Y 270.76,Z 787.756,A -85,B 0,C 180,E1 -17908.513,E2 -17908.513} C_VEL
LIN {X 0,Y 270.758,Z 787.756,A -85,B 0,C 180,E1 -17911.487,E2 -17911.487} C_VEL
LIN {X 0,Y 270.552,Z 787.781,A -85,B 0,C 180,E1 -17917.463,E2 -17917.463} C_VEL
LIN {X 0,Y 270.379,Z 787.805,A -85,B 0,C 180,E1 -17920.484,E2 -17920.484} C_VEL
LIN {X 0,Y 270.359,Z 787.805,A -85,B 0,C 180,E1 -17925.067,E2 -17925.067} C_VEL
LIN {X 0,Y 270.243,Z 787.819,A -85,B 0,C 180,E1 -17929.76,E2 -17929.76} C_VEL
LIN {X 0,Y 270.216,Z 787.826,A -85,B 0,C 180,E1 -17934.591,E2 -17934.591} C_VEL
LIN {X 0,Y 270.191,Z 787.826,A -85,B 0,C 180,E1 -17937.918,E2 -17937.918} C_VEL
LIN {X 0,Y 270.166,Z 787.829,A -85,B 0,C 180,E1 -17941.351,E2 -17941.351} C_VEL
LIN {X 0,Y 270.195,Z 787.83,A -85,B 0,C 180,E1 -17944.907,E2 -17944.907} C_VEL
LIN {X 0,Y 270.191,Z 787.828,A -85,B 0,C 180,E1 -17948.712,E2 -17948.712} C_VEL
LIN {X 0,Y 270.166,Z 787.829,A -85,B 0,C 180,E1 -17952.56,E2 -17952.56} C_VEL
LIN {X 0,Y 270.16,Z 787.831,A -85,B 0,C 180,E1 -17956.753,E2 -17956.753} C_VEL
LIN {X 0,Y 270.169,Z 787.832,A -85,B 0,C 180,E1 -17959.436,E2 -17959.436} C_VEL
LIN {X 0,Y 270.14,Z 787.835,A -85,B 0,C 180,E1 -17963.249,E2 -17963.249} C_VEL
LIN {X 0,Y 269.956,Z 787.855,A -85,B 0,C 180,E1 -17966.86,E2 -17966.86} C_VEL
LIN {X 0,Y 269.531,Z 787.908,A -85,B 0,C 180,E1 -17970.304,E2 -17970.304} C_VEL
LIN {X 0,Y 269.118,Z 787.964,A -85,B 0,C 180,E1 -17973.646,E2 -17973.646} C_VEL
LIN {X 0,Y 268.804,Z 788.202,A -85,B 0,C 180,E1 -17976.912,E2 -17976.912} C_VEL
LIN {X 0,Y 268.797,Z 788.386,A -85,B 0,C 180,E1 -17977.105,E2 -17977.105} C_VEL
LIN {X 0,Y 271.805,Z 804.067,A -85,B 0,C 180,E1 -17978.302,E2 -17978.302} C_VEL
LIN {X 0,Y 274.459,Z 817.881,A -85,B 0,C 180,E1 -17979.68,E2 -17979.68} C_VEL
LIN {X 0,Y 275.162,Z 822.59,A -85,B 0,C 180,E1 -17980.221,E2 -17980.221} C_VEL
LIN {X 0,Y 274.079,Z 834.211,A -85,B 0,C 180,E1 -17981.66,E2 -17981.66} C_VEL
LIN {X 0,Y 272.841,Z 845.265,A -85,B 0,C 180,E1 -17983.349,E2 -17983.349} C_VEL
LIN {X 0,Y 271.759,Z 854.285,A -85,B 0,C 180,E1 -17985.014,E2 -17985.014} C_VEL
LIN {X 0,Y 270.764,Z 862.677,A -85,B 0,C 180,E1 -17986.874,E2 -17986.874} C_VEL
LIN {X 0,Y 269.836,Z 870.951,A -85,B 0,C 180,E1 -17989.117,E2 -17989.117} C_VEL
LIN {X 0,Y 269.157,Z 877.711,A -85,B 0,C 180,E1 -17991.367,E2 -17991.367} C_VEL
LIN {X 0,Y 268.75,Z 883.083,A -85,B 0,C 180,E1 -17993.582,E2 -17993.582} C_VEL
LIN {X 0,Y 268.526,Z 888.046,A -85,B 0,C 180,E1 -17996.25,E2 -17996.25} C_VEL
LIN {X 0,Y 268.432,Z 891.113,A -85,B 0,C 180,E1 -17998.501,E2 -17998.501} C_VEL
LIN {X 0,Y 268.579,Z 893.708,A -85,B 0,C 180,E1 -18001.501,E2 -18001.501} C_VEL
LIN {X 0,Y 268.8,Z 894.394,A -85,B 0,C 180,E1 -18002.999,E2 -18002.999} C_VEL
LIN {X 0,Y 269.03,Z 894.667,A -85,B 0,C 180,E1 -18004.496,E2 -18004.496} C_VEL
LIN {X 0,Y 269.751,Z 894.088,A -85,B 0,C 180,E1 -18007.487,E2 -18007.487} C_VEL
LIN {X 0,Y 271.005,Z 892.523,A -85,B 0,C 180,E1 -18009.781,E2 -18009.781} C_VEL
LIN {X 0,Y 272.663,Z 889.23,A -85,B 0,C 180,E1 -18012.657,E2 -18012.657} C_VEL
LIN {X 0,Y 275.131,Z 884.215,A -85,B 0,C 180,E1 -18015.559,E2 -18015.559} C_VEL
LIN {X 0,Y 276.431,Z 881.39,A -85,B 0,C 180,E1 -18016.821,E2 -18016.821} C_VEL
LIN {X 0,Y 277.036,Z 878.943,A -85,B 0,C 180,E1 -18017.929,E2 -18017.929} C_VEL
LIN {X 0,Y 276.561,Z 874.975,A -85,B 0,C 180,E1 -18019.81,E2 -18019.81} C_VEL
LIN {X 0,Y 276.356,Z 870.457,A -85,B 0,C 180,E1 -18021.627,E2 -18021.627} C_VEL
LIN {X 0,Y 277.335,Z 867.159,A -85,B 0,C 180,E1 -18022.61,E2 -18022.61} C_VEL
LIN {X 0,Y 281.15,Z 858.033,A -85,B 0,C 180,E1 -18024.754,E2 -18024.754} C_VEL
LIN {X 0,Y 285.449,Z 846.819,A -85,B 0,C 180,E1 -18026.811,E2 -18026.811} C_VEL
LIN {X 0,Y 285.845,Z 845.669,A -85,B 0,C 180,E1 -18027.011,E2 -18027.011} C_VEL
LIN {X 0,Y 285.479,Z 839.687,A -85,B 0,C 180,E1 -18028.599,E2 -18028.599} C_VEL
LIN {X 0,Y 284.296,Z 833.587,A -85,B 0,C 180,E1 -18030.47,E2 -18030.47} C_VEL
LIN {X 0,Y 282.386,Z 827.243,A -85,B 0,C 180,E1 -18032.756,E2 -18032.756} C_VEL
LIN {X 0,Y 280.966,Z 823.574,A -85,B 0,C 180,E1 -18034.365,E2 -18034.365} C_VEL
LIN {X 0,Y 280.302,Z 821.859,A -85,B 0,C 180,E1 -18035.219,E2 -18035.219} C_VEL
LIN {X 0,Y 278.626,Z 818.666,A -85,B 0,C 180,E1 -18037.257,E2 -18037.257} C_VEL
LIN {X 0,Y 277.122,Z 816.608,A -85,B 0,C 180,E1 -18039.349,E2 -18039.349} C_VEL
LIN {X 0,Y 276.042,Z 814.729,A -85,B 0,C 180,E1 -18042.41,E2 -18042.41} C_VEL
LIN {X 0,Y 275.769,Z 814.738,A -85,B 0,C 180,E1 -18044.473,E2 -18044.473} C_VEL
LIN {X 0,Y 276.02,Z 815.732,A -85,B 0,C 180,E1 -18046.57,E2 -18046.57} C_VEL
LIN {X 0,Y 276.57,Z 818.119,A -85,B 0,C 180,E1 -18048.647,E2 -18048.647} C_VEL
LIN {X 0,Y 278.27,Z 822.559,A -85,B 0,C 180,E1 -18051.532,E2 -18051.532} C_VEL
LIN {X 0,Y 279.62,Z 828.662,A -85,B 0,C 180,E1 -18053.813,E2 -18053.813} C_VEL
LIN {X 0,Y 280.341,Z 836.279,A -85,B 0,C 180,E1 -18055.823,E2 -18055.823} C_VEL
LIN {X 0,Y 280.794,Z 845.729,A -85,B 0,C 180,E1 -18058.002,E2 -18058.002} C_VEL
LIN {X 0,Y 280.644,Z 857.169,A -85,B 0,C 180,E1 -18060.399,E2 -18060.399} C_VEL
LIN {X 0,Y 279.666,Z 867.225,A -85,B 0,C 180,E1 -18062.434,E2 -18062.434} C_VEL
LIN {X 0,Y 277.412,Z 877.481,A -85,B 0,C 180,E1 -18064.489,E2 -18064.489} C_VEL
LIN {X 0,Y 275.399,Z 884.096,A -85,B 0,C 180,E1 -18065.901,E2 -18065.901} C_VEL
LIN {X 0,Y 271.972,Z 892.914,A -85,B 0,C 180,E1 -18067.995,E2 -18067.995} C_VEL
LIN {X 0,Y 269.041,Z 900.344,A -85,B 0,C 180,E1 -18070.148,E2 -18070.148} C_VEL
LIN {X 0,Y 266.628,Z 906.543,A -85,B 0,C 180,E1 -18072.354,E2 -18072.354} C_VEL
LIN {X 0,Y 264.131,Z 913.205,A -85,B 0,C 180,E1 -18075.358,E2 -18075.358} C_VEL
LIN {X 0,Y 262.765,Z 917.014,A -85,B 0,C 180,E1 -18077.645,E2 -18077.645} C_VEL
LIN {X 0,Y 262.167,Z 919.075,A -85,B 0,C 180,E1 -18079.184,E2 -18079.184} C_VEL
LIN {X 0,Y 261.405,Z 921.935,A -85,B 0,C 180,E1 -18082.274,E2 -18082.274} C_VEL
LIN {X 0,Y 261.35,Z 922.989,A -85,B 0,C 180,E1 -18084.263,E2 -18084.263} C_VEL
LIN {X 0,Y 261.338,Z 923.307,A -85,B 0,C 180,E1 -18086.917,E2 -18086.917} C_VEL
LIN {X 0,Y 261.681,Z 922.84,A -85,B 0,C 180,E1 -18088.846,E2 -18088.846} C_VEL
LIN {X 0,Y 261.717,Z 923.714,A -85,B 0,C 180,E1 -18090,E2 -18090} C_VEL
LIN {X 0,Y 261.287,Z 924.814,A -85,B 0,C 180,E1 -18093.084,E2 -18093.084} C_VEL
LIN {X 0,Y 261.225,Z 924.551,A -85,B 0,C 180,E1 -18095.458,E2 -18095.458} C_VEL
LIN {X 0,Y 261.383,Z 923.426,A -85,B 0,C 180,E1 -18097.726,E2 -18097.726} C_VEL
LIN {X 0,Y 262.138,Z 920.582,A -85,B 0,C 180,E1 -18100.817,E2 -18100.817} C_VEL
LIN {X 0,Y 263.121,Z 917.379,A -85,B 0,C 180,E1 -18103.123,E2 -18103.123} C_VEL
LIN {X 0,Y 264.752,Z 913.269,A -85,B 0,C 180,E1 -18105.394,E2 -18105.394} C_VEL
LIN {X 0,Y 266.674,Z 908.19,A -85,B 0,C 180,E1 -18107.642,E2 -18107.642} C_VEL
LIN {X 0,Y 269.004,Z 902.054,A -85,B 0,C 180,E1 -18109.855,E2 -18109.855} C_VEL
LIN {X 0,Y 271.908,Z 894.772,A -85,B 0,C 180,E1 -18112.011,E2 -18112.011} C_VEL
LIN {X 0,Y 276.108,Z 884.467,A -85,B 0,C 180,E1 -18114.433,E2 -18114.433} C_VEL
LIN {X 0,Y 278.227,Z 877.829,A -85,B 0,C 180,E1 -18115.832,E2 -18115.832} C_VEL
LIN {X 0,Y 280.029,Z 870.128,A -85,B 0,C 180,E1 -18117.355,E2 -18117.355} C_VEL
LIN {X 0,Y 280.859,Z 862.928,A -85,B 0,C 180,E1 -18118.856,E2 -18118.856} C_VEL
LIN {X 0,Y 281.014,Z 853.527,A -85,B 0,C 180,E1 -18120.899,E2 -18120.899} C_VEL
LIN {X 0,Y 280.455,Z 845.852,A -85,B 0,C 180,E1 -18122.737,E2 -18122.737} C_VEL
LIN {X 0,Y 279.356,Z 837.488,A -85,B 0,C 180,E1 -18125.028,E2 -18125.028} C_VEL
LIN {X 0,Y 278.451,Z 832.468,A -85,B 0,C 180,E1 -18126.647,E2 -18126.647} C_VEL
LIN {X 0,Y 277.619,Z 828.02,A -85,B 0,C 180,E1 -18128.299,E2 -18128.299} C_VEL
LIN {X 0,Y 275.862,Z 822.859,A -85,B 0,C 180,E1 -18131.483,E2 -18131.483} C_VEL
LIN {X 0,Y 275.427,Z 820.256,A -85,B 0,C 180,E1 -18133.547,E2 -18133.547} C_VEL
LIN {X 0,Y 275.251,Z 819.045,A -85,B 0,C 180,E1 -18135.637,E2 -18135.637} C_VEL
LIN {X 0,Y 275.457,Z 819.052,A -85,B 0,C 180,E1 -18137.724,E2 -18137.724} C_VEL
LIN {X 0,Y 276.514,Z 820.306,A -85,B 0,C 180,E1 -18140.548,E2 -18140.548} C_VEL
LIN {X 0,Y 277.976,Z 821.953,A -85,B 0,C 180,E1 -18142.641,E2 -18142.641} C_VEL
LIN {X 0,Y 279.656,Z 824.656,A -85,B 0,C 180,E1 -18144.688,E2 -18144.688} C_VEL
LIN {X 0,Y 281.867,Z 829.701,A -85,B 0,C 180,E1 -18147.255,E2 -18147.255} C_VEL
LIN {X 0,Y 283.527,Z 834.371,A -85,B 0,C 180,E1 -18149.143,E2 -18149.143} C_VEL
LIN {X 0,Y 285.042,Z 840.087,A -85,B 0,C 180,E1 -18151.09,E2 -18151.09} C_VEL
LIN {X 0,Y 285.982,Z 846.493,A -85,B 0,C 180,E1 -18152.999,E2 -18152.999} C_VEL
LIN {X 0,Y 284.861,Z 849.971,A -85,B 0,C 180,E1 -18153.633,E2 -18153.633} C_VEL
LIN {X 0,Y 280.839,Z 860.214,A -85,B 0,C 180,E1 -18155.611,E2 -18155.611} C_VEL
LIN {X 0,Y 277.117,Z 868.651,A -85,B 0,C 180,E1 -18157.639,E2 -18157.639} C_VEL
LIN {X 0,Y 273.348,Z 876.742,A -85,B 0,C 180,E1 -18160.081,E2 -18160.081} C_VEL
LIN {X 0,Y 270.242,Z 883.116,A -85,B 0,C 180,E1 -18162.597,E2 -18162.597} C_VEL
LIN {X 0,Y 267.887,Z 887.51,A -85,B 0,C 180,E1 -18164.789,E2 -18164.789} C_VEL
LIN {X 0,Y 265.4,Z 891.804,A -85,B 0,C 180,E1 -18167.768,E2 -18167.768} C_VEL
LIN {X 0,Y 264.299,Z 893.698,A -85,B 0,C 180,E1 -18169.697,E2 -18169.697} C_VEL
LIN {X 0,Y 262.79,Z 895.306,A -85,B 0,C 180,E1 -18172.314,E2 -18172.314} C_VEL
LIN {X 0,Y 262.089,Z 895.699,A -85,B 0,C 180,E1 -18175.384,E2 -18175.384} C_VEL
LIN {X 0,Y 261.784,Z 895.329,A -85,B 0,C 180,E1 -18176.921,E2 -18176.921} C_VEL
LIN {X 0,Y 261.411,Z 893.367,A -85,B 0,C 180,E1 -18179.998,E2 -18179.998} C_VEL
LIN {X 0,Y 261.394,Z 890.842,A -85,B 0,C 180,E1 -18182.31,E2 -18182.31} C_VEL
LIN {X 0,Y 261.511,Z 887.349,A -85,B 0,C 180,E1 -18184.623,E2 -18184.623} C_VEL
LIN {X 0,Y 261.772,Z 882.782,A -85,B 0,C 180,E1 -18186.937,E2 -18186.937} C_VEL
LIN {X 0,Y 262.34,Z 875.949,A -85,B 0,C 180,E1 -18189.637,E2 -18189.637} C_VEL
LIN {X 0,Y 263.16,Z 868.563,A -85,B 0,C 180,E1 -18191.943,E2 -18191.943} C_VEL
LIN {X 0,Y 264.184,Z 859.525,A -85,B 0,C 180,E1 -18194.244,E2 -18194.244} C_VEL
LIN {X 0,Y 265.417,Z 849.391,A -85,B 0,C 180,E1 -18196.338,E2 -18196.338} C_VEL
LIN {X 0,Y 266.684,Z 839.36,A -85,B 0,C 180,E1 -18198.036,E2 -18198.036} C_VEL
LIN {X 0,Y 267.979,Z 827.122,A -85,B 0,C 180,E1 -18199.732,E2 -18199.732} C_VEL
LIN {X 0,Y 268.129,Z 822.215,A -85,B 0,C 180,E1 -18200.32,E2 -18200.32} C_VEL
LIN {X 0,Y 265.402,Z 808.174,A -85,B 0,C 180,E1 -18201.846,E2 -18201.846} C_VEL
LIN {X 0,Y 262.714,Z 794.573,A -85,B 0,C 180,E1 -18203.001,E2 -18203.001} C_VEL
LIN {X 0,Y 261.812,Z 789.627,A -85,B 0,C 180,E1 -18203.399,E2 -18203.399} C_VEL
LIN {X 0,Y 261.823,Z 789.04,A -85,B 0,C 180,E1 -18204.126,E2 -18204.126} C_VEL
LIN {X 0,Y 262.213,Z 788.823,A -85,B 0,C 180,E1 -18207.811,E2 -18207.811} C_VEL
LIN {X 0,Y 262.575,Z 788.773,A -85,B 0,C 180,E1 -18211.074,E2 -18211.074} C_VEL
LIN {X 0,Y 262.907,Z 788.735,A -85,B 0,C 180,E1 -18214.148,E2 -18214.148} C_VEL
LIN {X 0,Y 263.061,Z 788.714,A -85,B 0,C 180,E1 -18217.911,E2 -18217.911} C_VEL
LIN {X 0,Y 263.119,Z 788.706,A -85,B 0,C 180,E1 -18221.892,E2 -18221.892} C_VEL
LIN {X 0,Y 263.099,Z 788.71,A -85,B 0,C 180,E1 -18226.154,E2 -18226.154} C_VEL
LIN {X 0,Y 263.099,Z 788.708,A -85,B 0,C 180,E1 -18230.126,E2 -18230.126} C_VEL
LIN {X 0,Y 263.156,Z 788.702,A -85,B 0,C 180,E1 -18234.017,E2 -18234.017} C_VEL
LIN {X 0,Y 263.121,Z 788.705,A -85,B 0,C 180,E1 -18237.71,E2 -18237.71} C_VEL
LIN {X 0,Y 263.141,Z 788.705,A -85,B 0,C 180,E1 -18241.804,E2 -18241.804} C_VEL
LIN {X 0,Y 263.182,Z 788.703,A -85,B 0,C 180,E1 -18245.217,E2 -18245.217} C_VEL
LIN {X 0,Y 263.227,Z 788.696,A -85,B 0,C 180,E1 -18249.69,E2 -18249.69} C_VEL
LIN {X 0,Y 263.302,Z 788.683,A -85,B 0,C 180,E1 -18254.519,E2 -18254.519} C_VEL
LIN {X 0,Y 263.344,Z 788.68,A -85,B 0,C 180,E1 -18259.233,E2 -18259.233} C_VEL
LIN {X 0,Y 263.516,Z 788.658,A -85,B 0,C 180,E1 -18262.337,E2 -18262.337} C_VEL
LIN {X 0,Y 263.723,Z 788.633,A -85,B 0,C 180,E1 -18268.473,E2 -18268.473} C_VEL
LIN {X 0,Y 263.721,Z 788.633,A -85,B 0,C 180,E1 -18271.527,E2 -18271.527} C_VEL
LIN {X 0,Y 263.516,Z 788.658,A -85,B 0,C 180,E1 -18277.663,E2 -18277.663} C_VEL
LIN {X 0,Y 263.325,Z 788.682,A -85,B 0,C 180,E1 -18280.768,E2 -18280.768} C_VEL
LIN {X 0,Y 263.302,Z 788.683,A -85,B 0,C 180,E1 -18285.481,E2 -18285.481} C_VEL
LIN {X 0,Y 263.227,Z 788.696,A -85,B 0,C 180,E1 -18290.31,E2 -18290.31} C_VEL
LIN {X 0,Y 263.159,Z 788.703,A -85,B 0,C 180,E1 -18295.296,E2 -18295.296} C_VEL
LIN {X 0,Y 263.126,Z 788.711,A -85,B 0,C 180,E1 -18298.736,E2 -18298.736} C_VEL
LIN {X 0,Y 263.121,Z 788.705,A -85,B 0,C 180,E1 -18302.29,E2 -18302.29} C_VEL
LIN {X 0,Y 263.175,Z 788.703,A -85,B 0,C 180,E1 -18306.764,E2 -18306.764} C_VEL
LIN {X 0,Y 263.119,Z 788.708,A -85,B 0,C 180,E1 -18311.595,E2 -18311.595} C_VEL
LIN {X 0,Y 263.1,Z 788.709,A -85,B 0,C 180,E1 -18316.157,E2 -18316.157} C_VEL
LIN {X 0,Y 263.101,Z 788.708,A -85,B 0,C 180,E1 -18320.129,E2 -18320.129} C_VEL
LIN {X 0,Y 263.051,Z 788.717,A -85,B 0,C 180,E1 -18324.003,E2 -18324.003} C_VEL
LIN {X 0,Y 262.788,Z 788.75,A -85,B 0,C 180,E1 -18327.666,E2 -18327.666} C_VEL
LIN {X 0,Y 262.367,Z 788.801,A -85,B 0,C 180,E1 -18331.175,E2 -18331.175} C_VEL
LIN {X 0,Y 261.953,Z 788.852,A -85,B 0,C 180,E1 -18334.581,E2 -18334.581} C_VEL
LIN {X 0,Y 261.758,Z 788.882,A -85,B 0,C 180,E1 -18336.829,E2 -18336.829} C_VEL
LIN {X 0,Y 264.635,Z 804.092,A -85,B 0,C 180,E1 -18338.006,E2 -18338.006} C_VEL
LIN {X 0,Y 267.369,Z 818.28,A -85,B 0,C 180,E1 -18339.451,E2 -18339.451} C_VEL
LIN {X 0,Y 268.106,Z 823.612,A -85,B 0,C 180,E1 -18340.078,E2 -18340.078} C_VEL
LIN {X 0,Y 266.917,Z 835.226,A -85,B 0,C 180,E1 -18341.583,E2 -18341.583} C_VEL
LIN {X 0,Y 265.853,Z 844.833,A -85,B 0,C 180,E1 -18343.096,E2 -18343.096} C_VEL
LIN {X 0,Y 264.646,Z 854.87,A -85,B 0,C 180,E1 -18344.996,E2 -18344.996} C_VEL
LIN {X 0,Y 263.47,Z 864.695,A -85,B 0,C 180,E1 -18347.289,E2 -18347.289} C_VEL
LIN {X 0,Y 262.575,Z 872.734,A -85,B 0,C 180,E1 -18349.593,E2 -18349.593} C_VEL
LIN {X 0,Y 262.042,Z 878.248,A -85,B 0,C 180,E1 -18351.519,E2 -18351.519} C_VEL
LIN {X 0,Y 261.64,Z 883.704,A -85,B 0,C 180,E1 -18353.834,E2 -18353.834} C_VEL
LIN {X 0,Y 261.443,Z 887.966,A -85,B 0,C 180,E1 -18356.148,E2 -18356.148} C_VEL
LIN {X 0,Y 261.353,Z 891.18,A -85,B 0,C 180,E1 -18358.461,E2 -18358.461} C_VEL
LIN {X 0,Y 261.368,Z 892.771,A -85,B 0,C 180,E1 -18360.002,E2 -18360.002} C_VEL
LIN {X 0,Y 261.723,Z 894.769,A -85,B 0,C 180,E1 -18363.08,E2 -18363.08} C_VEL
LIN {X 0,Y 261.968,Z 895.18,A -85,B 0,C 180,E1 -18364.618,E2 -18364.618} C_VEL
LIN {X 0,Y 262.766,Z 894.794,A -85,B 0,C 180,E1 -18367.687,E2 -18367.687} C_VEL
LIN {X 0,Y 264.02,Z 893.472,A -85,B 0,C 180,E1 -18369.964,E2 -18369.964} C_VEL
LIN {X 0,Y 265.321,Z 891.31,A -85,B 0,C 180,E1 -18372.236,E2 -18372.236} C_VEL
LIN {X 0,Y 267.706,Z 887.039,A -85,B 0,C 180,E1 -18375.222,E2 -18375.222} C_VEL
LIN {X 0,Y 270.911,Z 880.925,A -85,B 0,C 180,E1 -18378.139,E2 -18378.139} C_VEL
LIN {X 0,Y 274.125,Z 874.09,A -85,B 0,C 180,E1 -18380.643,E2 -18380.643} C_VEL
LIN {X 0,Y 277.335,Z 867.159,A -85,B 0,C 180,E1 -18382.61,E2 -18382.61} C_VEL
LIN {X 0,Y 278.778,Z 862.565,A -85,B 0,C 180,E1 -18383.884,E2 -18383.884} C_VEL
LIN {X 0,Y 279.282,Z 858.145,A -85,B 0,C 180,E1 -18385.218,E2 -18385.218} C_VEL
LIN {X 0,Y 279.544,Z 853.588,A -85,B 0,C 180,E1 -18386.547,E2 -18386.547} C_VEL
LIN {X 0,Y 280.241,Z 848.574,A -85,B 0,C 180,E1 -18387.79,E2 -18387.79} C_VEL
LIN {X 0,Y 280.437,Z 846.095,A -85,B 0,C 180,E1 -18388.436,E2 -18388.436} C_VEL
LIN {X 0,Y 279.91,Z 840.585,A -85,B 0,C 180,E1 -18390.145,E2 -18390.145} C_VEL
LIN {X 0,Y 278.42,Z 833.547,A -85,B 0,C 180,E1 -18392.737,E2 -18392.737} C_VEL
LIN {X 0,Y 277.1,Z 829.354,A -85,B 0,C 180,E1 -18394.652,E2 -18394.652} C_VEL
LIN {X 0,Y 275.794,Z 826.113,A -85,B 0,C 180,E1 -18396.559,E2 -18396.559} C_VEL
LIN {X 0,Y 274.972,Z 824.421,A -85,B 0,C 180,E1 -18397.838,E2 -18397.838} C_VEL
LIN {X 0,Y 273.815,Z 822.681,A -85,B 0,C 180,E1 -18399.918,E2 -18399.918} C_VEL
LIN {X 0,Y 273.209,Z 821.472,A -85,B 0,C 180,E1 -18401.978,E2 -18401.978} C_VEL
LIN {X 0,Y 272.999,Z 821.165,A -85,B 0,C 180,E1 -18404.035,E2 -18404.035} C_VEL
LIN {X 0,Y 273.082,Z 822.009,A -85,B 0,C 180,E1 -18406.106,E2 -18406.106} C_VEL
LIN {X 0,Y 273.472,Z 824.149,A -85,B 0,C 180,E1 -18408.185,E2 -18408.185} C_VEL
LIN {X 0,Y 274.329,Z 826.979,A -85,B 0,C 180,E1 -18410.227,E2 -18410.227} C_VEL
LIN {X 0,Y 275.091,Z 829.847,A -85,B 0,C 180,E1 -18411.713,E2 -18411.713} C_VEL
LIN {X 0,Y 275.697,Z 834.044,A -85,B 0,C 180,E1 -18413.283,E2 -18413.283} C_VEL
LIN {X 0,Y 275.94,Z 841.081,A -85,B 0,C 180,E1 -18415.224,E2 -18415.224} C_VEL
LIN {X 0,Y 275.822,Z 851.112,A -85,B 0,C 180,E1 -18417.65,E2 -18417.65} C_VEL
LIN {X 0,Y 274.99,Z 862.494,A -85,B 0,C 180,E1 -18420.192,E2 -18420.192} C_VEL
LIN {X 0,Y 273.489,Z 871.785,A -85,B 0,C 180,E1 -18422.195,E2 -18422.195} C_VEL
LIN {X 0,Y 270.344,Z 882.754,A -85,B 0,C 180,E1 -18424.599,E2 -18424.599} C_VEL
LIN {X 0,Y 266.099,Z 892.919,A -85,B 0,C 180,E1 -18427.072,E2 -18427.072} C_VEL
LIN {X 0,Y 262.442,Z 901.271,A -85,B 0,C 180,E1 -18429.627,E2 -18429.627} C_VEL
LIN {X 0,Y 259.908,Z 907.205,A -85,B 0,C 180,E1 -18431.883,E2 -18431.883} C_VEL
LIN {X 0,Y 257.903,Z 912.073,A -85,B 0,C 180,E1 -18434.187,E2 -18434.187} C_VEL
LIN {X 0,Y 256.214,Z 916.004,A -85,B 0,C 180,E1 -18436.517,E2 -18436.517} C_VEL
LIN {X 0,Y 255.156,Z 919.013,A -85,B 0,C 180,E1 -18438.883,E2 -18438.883} C_VEL
LIN {X 0,Y 254.35,Z 921.686,A -85,B 0,C 180,E1 -18442.059,E2 -18442.059} C_VEL
LIN {X 0,Y 254.259,Z 922.616,A -85,B 0,C 180,E1 -18444.325,E2 -18444.325} C_VEL
LIN {X 0,Y 254.266,Z 922.716,A -85,B 0,C 180,E1 -18446.831,E2 -18446.831} C_VEL
LIN {X 0,Y 254.631,Z 922.154,A -85,B 0,C 180,E1 -18449.012,E2 -18449.012} C_VEL
LIN {X 0,Y 254.661,Z 922.94,A -85,B 0,C 180,E1 -18450,E2 -18450} C_VEL
LIN {X 0,Y 254.215,Z 924.206,A -85,B 0,C 180,E1 -18453.17,E2 -18453.17} C_VEL
LIN {X 0,Y 254.139,Z 924.161,A -85,B 0,C 180,E1 -18455.396,E2 -18455.396} C_VEL
LIN {X 0,Y 254.333,Z 923.162,A -85,B 0,C 180,E1 -18457.942,E2 -18457.942} C_VEL
LIN {X 0,Y 255.131,Z 920.495,A -85,B 0,C 180,E1 -18461.118,E2 -18461.118} C_VEL
LIN {X 0,Y 256.666,Z 916.346,A -85,B 0,C 180,E1 -18464.267,E2 -18464.267} C_VEL
LIN {X 0,Y 258.564,Z 912.118,A -85,B 0,C 180,E1 -18466.583,E2 -18466.583} C_VEL
LIN {X 0,Y 261.345,Z 905.305,A -85,B 0,C 180,E1 -18469.534,E2 -18469.534} C_VEL
LIN {X 0,Y 264.88,Z 897.242,A -85,B 0,C 180,E1 -18472.216,E2 -18472.216} C_VEL
LIN {X 0,Y 269.156,Z 887.766,A -85,B 0,C 180,E1 -18474.695,E2 -18474.695} C_VEL
LIN {X 0,Y 271.625,Z 881.5,A -85,B 0,C 180,E1 -18476.095,E2 -18476.095} C_VEL
LIN {X 0,Y 274.288,Z 872.177,A -85,B 0,C 180,E1 -18478.109,E2 -18478.109} C_VEL
LIN {X 0,Y 275.358,Z 864.558,A -85,B 0,C 180,E1 -18479.795,E2 -18479.795} C_VEL
LIN {X 0,Y 275.76,Z 854.895,A -85,B 0,C 180,E1 -18482.09,E2 -18482.09} C_VEL
LIN {X 0,Y 275.42,Z 847.182,A -85,B 0,C 180,E1 -18484.152,E2 -18484.152} C_VEL
LIN {X 0,Y 274.664,Z 839.193,A -85,B 0,C 180,E1 -18486.642,E2 -18486.642} C_VEL
LIN {X 0,Y 273.833,Z 833.432,A -85,B 0,C 180,E1 -18488.927,E2 -18488.927} C_VEL
LIN {X 0,Y 272.552,Z 828.553,A -85,B 0,C 180,E1 -18492.101,E2 -18492.101} C_VEL
LIN {X 0,Y 272.345,Z 826.306,A -85,B 0,C 180,E1 -18494.167,E2 -18494.167} C_VEL
LIN {X 0,Y 272.316,Z 825.378,A -85,B 0,C 180,E1 -18496.272,E2 -18496.272} C_VEL
LIN {X 0,Y 272.526,Z 825.715,A -85,B 0,C 180,E1 -18498.406,E2 -18498.406} C_VEL
LIN {X 0,Y 273.299,Z 826.633,A -85,B 0,C 180,E1 -18500.486,E2 -18500.486} C_VEL
LIN {X 0,Y 274.536,Z 828.138,A -85,B 0,C 180,E1 -18502.522,E2 -18502.522} C_VEL
LIN {X 0,Y 275.966,Z 830.783,A -85,B 0,C 180,E1 -18504.582,E2 -18504.582} C_VEL
LIN {X 0,Y 277.466,Z 834.676,A -85,B 0,C 180,E1 -18506.706,E2 -18506.706} C_VEL
LIN {X 0,Y 279.236,Z 840.817,A -85,B 0,C 180,E1 -18509.327,E2 -18509.327} C_VEL
LIN {X 0,Y 280.261,Z 847.24,A -85,B 0,C 180,E1 -18511.544,E2 -18511.544} C_VEL
LIN {X 0,Y 280.481,Z 849.882,A -85,B 0,C 180,E1 -18512.369,E2 -18512.369} C_VEL
LIN {X 0,Y 276.145,Z 860.109,A -85,B 0,C 180,E1 -18514.362,E2 -18514.362} C_VEL
LIN {X 0,Y 271.513,Z 869.898,A -85,B 0,C 180,E1 -18516.749,E2 -18516.749} C_VEL
LIN {X 0,Y 267.449,Z 877.777,A -85,B 0,C 180,E1 -18519.22,E2 -18519.22} C_VEL
LIN {X 0,Y 264.56,Z 883.24,A -85,B 0,C 180,E1 -18521.409,E2 -18521.409} C_VEL
LIN {X 0,Y 261.975,Z 887.664,A -85,B 0,C 180,E1 -18523.638,E2 -18523.638} C_VEL
LIN {X 0,Y 259.799,Z 891.12,A -85,B 0,C 180,E1 -18525.907,E2 -18525.907} C_VEL
LIN {X 0,Y 258.562,Z 892.948,A -85,B 0,C 180,E1 -18527.439,E2 -18527.439} C_VEL
LIN {X 0,Y 256.753,Z 895.345,A -85,B 0,C 180,E1 -18530.546,E2 -18530.546} C_VEL
LIN {X 0,Y 255.81,Z 896.028,A -85,B 0,C 180,E1 -18532.103,E2 -18532.103} C_VEL
LIN {X 0,Y 255.322,Z 896.314,A -85,B 0,C 180,E1 -18533.677,E2 -18533.677} C_VEL
LIN {X 0,Y 255.025,Z 896.182,A -85,B 0,C 180,E1 -18535.256,E2 -18535.256} C_VEL
LIN {X 0,Y 254.456,Z 894.798,A -85,B 0,C 180,E1 -18538.416,E2 -18538.416} C_VEL
LIN {X 0,Y 254.327,Z 893.537,A -85,B 0,C 180,E1 -18539.998,E2 -18539.998} C_VEL
LIN {X 0,Y 254.322,Z 890.831,A -85,B 0,C 180,E1 -18542.374,E2 -18542.374} C_VEL
LIN {X 0,Y 254.42,Z 887.149,A -85,B 0,C 180,E1 -18544.752,E2 -18544.752} C_VEL
LIN {X 0,Y 254.788,Z 881.239,A -85,B 0,C 180,E1 -18547.626,E2 -18547.626} C_VEL
LIN {X 0,Y 255.435,Z 874.169,A -85,B 0,C 180,E1 -18550.3,E2 -18550.3} C_VEL
LIN {X 0,Y 256.346,Z 866.328,A -85,B 0,C 180,E1 -18552.668,E2 -18552.668} C_VEL
LIN {X 0,Y 257.511,Z 856.634,A -85,B 0,C 180,E1 -18555.025,E2 -18555.025} C_VEL
LIN {X 0,Y 258.694,Z 846.857,A -85,B 0,C 180,E1 -18556.979,E2 -18556.979} C_VEL
LIN {X 0,Y 259.725,Z 838.373,A -85,B 0,C 180,E1 -18558.393,E2 -18558.393} C_VEL
LIN {X 0,Y 261.062,Z 826.212,A -85,B 0,C 180,E1 -18560.072,E2 -18560.072} C_VEL
LIN {X 0,Y 261.026,Z 822.899,A -85,B 0,C 180,E1 -18560.487,E2 -18560.487} C_VEL
LIN {X 0,Y 258.305,Z 808.633,A -85,B 0,C 180,E1 -18562.089,E2 -18562.089} C_VEL
LIN {X 0,Y 255.642,Z 794.937,A -85,B 0,C 180,E1 -18563.289,E2 -18563.289} C_VEL
LIN {X 0,Y 254.738,Z 790.048,A -85,B 0,C 180,E1 -18563.687,E2 -18563.687} C_VEL
LIN {X 0,Y 254.79,Z 789.753,A -85,B 0,C 180,E1 -18564.459,E2 -18564.459} C_VEL
LIN {X 0,Y 255.211,Z 789.696,A -85,B 0,C 180,E1 -18568.21,E2 -18568.21} C_VEL
LIN {X 0,Y 255.576,Z 789.644,A -85,B 0,C 180,E1 -18571.52,E2 -18571.52} C_VEL
LIN {X 0,Y 255.901,Z 789.606,A -85,B 0,C 180,E1 -18575.219,E2 -18575.219} C_VEL
LIN {X 0,Y 256.003,Z 789.594,A -85,B 0,C 180,E1 -18577.238,E2 -18577.238} C_VEL
LIN {X 0,Y 256.048,Z 789.587,A -85,B 0,C 180,E1 -18581.202,E2 -18581.202} C_VEL
LIN {X 0,Y 256.036,Z 789.59,A -85,B 0,C 180,E1 -18585.533,E2 -18585.533} C_VEL
LIN {X 0,Y 256.049,Z 789.59,A -85,B 0,C 180,E1 -18588.795,E2 -18588.795} C_VEL
LIN {X 0,Y 256.123,Z 789.582,A -85,B 0,C 180,E1 -18592.866,E2 -18592.866} C_VEL
LIN {X 0,Y 256.059,Z 789.588,A -85,B 0,C 180,E1 -18596.706,E2 -18596.706} C_VEL
LIN {X 0,Y 256.047,Z 789.587,A -85,B 0,C 180,E1 -18600.392,E2 -18600.392} C_VEL
LIN {X 0,Y 256.125,Z 789.58,A -85,B 0,C 180,E1 -18604.887,E2 -18604.887} C_VEL
LIN {X 0,Y 256.139,Z 789.577,A -85,B 0,C 180,E1 -18609.102,E2 -18609.102} C_VEL
LIN {X 0,Y 256.222,Z 789.566,A -85,B 0,C 180,E1 -18614.08,E2 -18614.08} C_VEL
LIN {X 0,Y 256.278,Z 789.559,A -85,B 0,C 180,E1 -18617.327,E2 -18617.327} C_VEL
LIN {X 0,Y 256.426,Z 789.541,A -85,B 0,C 180,E1 -18620.622,E2 -18620.622} C_VEL
LIN {X 0,Y 256.444,Z 789.542,A -85,B 0,C 180,E1 -18623.706,E2 -18623.706} C_VEL
LIN {X 0,Y 256.686,Z 789.51,A -85,B 0,C 180,E1 -18628.431,E2 -18628.431} C_VEL
LIN {X 0,Y 256.684,Z 789.51,A -85,B 0,C 180,E1 -18631.569,E2 -18631.569} C_VEL
LIN {X 0,Y 256.443,Z 789.542,A -85,B 0,C 180,E1 -18636.294,E2 -18636.294} C_VEL
LIN {X 0,Y 256.393,Z 789.545,A -85,B 0,C 180,E1 -18639.466,E2 -18639.466} C_VEL
LIN {X 0,Y 256.223,Z 789.567,A -85,B 0,C 180,E1 -18644.292,E2 -18644.292} C_VEL
LIN {X 0,Y 256.16,Z 789.574,A -85,B 0,C 180,E1 -18647.566,E2 -18647.566} C_VEL
LIN {X 0,Y 256.133,Z 789.577,A -85,B 0,C 180,E1 -18651.111,E2 -18651.111} C_VEL
LIN {X 0,Y 256.125,Z 789.58,A -85,B 0,C 180,E1 -18655.113,E2 -18655.113} C_VEL
LIN {X 0,Y 256.047,Z 789.587,A -85,B 0,C 180,E1 -18659.608,E2 -18659.608} C_VEL
LIN {X 0,Y 256.059,Z 789.588,A -85,B 0,C 180,E1 -18663.294,E2 -18663.294} C_VEL
LIN {X 0,Y 256.108,Z 789.583,A -85,B 0,C 180,E1 -18667.272,E2 -18667.272} C_VEL
LIN {X 0,Y 256.049,Z 789.59,A -85,B 0,C 180,E1 -18671.205,E2 -18671.205} C_VEL
LIN {X 0,Y 256.036,Z 789.592,A -85,B 0,C 180,E1 -18675.536,E2 -18675.536} C_VEL
LIN {X 0,Y 256.05,Z 789.587,A -85,B 0,C 180,E1 -18678.798,E2 -18678.798} C_VEL
LIN {X 0,Y 256.062,Z 789.586,A -85,B 0,C 180,E1 -18682.858,E2 -18682.858} C_VEL
LIN {X 0,Y 255.834,Z 789.614,A -85,B 0,C 180,E1 -18686.675,E2 -18686.675} C_VEL
LIN {X 0,Y 255.415,Z 789.667,A -85,B 0,C 180,E1 -18690.313,E2 -18690.313} C_VEL
LIN {X 0,Y 254.998,Z 789.723,A -85,B 0,C 180,E1 -18693.836,E2 -18693.836} C_VEL
LIN {X 0,Y 254.756,Z 789.753,A -85,B 0,C 180,E1 -18696.571,E2 -18696.571} C_VEL
LIN {X 0,Y 257.586,Z 804.732,A -85,B 0,C 180,E1 -18697.777,E2 -18697.777} C_VEL
LIN {X 0,Y 260.36,Z 819.202,A -85,B 0,C 180,E1 -18699.306,E2 -18699.306} C_VEL
LIN {X 0,Y 260.996,Z 824.603,A -85,B 0,C 180,E1 -18699.963,E2 -18699.963} C_VEL
LIN {X 0,Y 259.727,Z 836.545,A -85,B 0,C 180,E1 -18701.576,E2 -18701.576} C_VEL
LIN {X 0,Y 258.696,Z 845.399,A -85,B 0,C 180,E1 -18703.021,E2 -18703.021} C_VEL
LIN {X 0,Y 257.515,Z 855.427,A -85,B 0,C 180,E1 -18704.975,E2 -18704.975} C_VEL
LIN {X 0,Y 256.347,Z 865.241,A -85,B 0,C 180,E1 -18707.332,E2 -18707.332} C_VEL
LIN {X 0,Y 255.422,Z 873.25,A -85,B 0,C 180,E1 -18709.699,E2 -18709.699} C_VEL
LIN {X 0,Y 254.833,Z 879.72,A -85,B 0,C 180,E1 -18712.076,E2 -18712.076} C_VEL
LIN {X 0,Y 254.432,Z 884.9,A -85,B 0,C 180,E1 -18714.441,E2 -18714.441} C_VEL
LIN {X 0,Y 254.325,Z 889.015,A -85,B 0,C 180,E1 -18716.833,E2 -18716.833} C_VEL
LIN {X 0,Y 254.276,Z 891.168,A -85,B 0,C 180,E1 -18718.418,E2 -18718.418} C_VEL
LIN {X 0,Y 254.286,Z 892.915,A -85,B 0,C 180,E1 -18720.002,E2 -18720.002} C_VEL
LIN {X 0,Y 254.416,Z 894.208,A -85,B 0,C 180,E1 -18721.585,E2 -18721.585} C_VEL
LIN {X 0,Y 254.65,Z 895.101,A -85,B 0,C 180,E1 -18723.166,E2 -18723.166} C_VEL
LIN {X 0,Y 255.229,Z 895.777,A -85,B 0,C 180,E1 -18726.325,E2 -18726.325} C_VEL
LIN {X 0,Y 255.787,Z 895.499,A -85,B 0,C 180,E1 -18727.898,E2 -18727.898} C_VEL
LIN {X 0,Y 257.101,Z 894.384,A -85,B 0,C 180,E1 -18730.235,E2 -18730.235} C_VEL
LIN {X 0,Y 258.472,Z 892.435,A -85,B 0,C 180,E1 -18732.565,E2 -18732.565} C_VEL
LIN {X 0,Y 260.989,Z 888.401,A -85,B 0,C 180,E1 -18735.623,E2 -18735.623} C_VEL
LIN {X 0,Y 263.438,Z 884.295,A -85,B 0,C 180,E1 -18737.868,E2 -18737.868} C_VEL
LIN {X 0,Y 266.301,Z 879.116,A -85,B 0,C 180,E1 -18740.066,E2 -18740.066} C_VEL
LIN {X 0,Y 269.513,Z 872.893,A -85,B 0,C 180,E1 -18742.218,E2 -18742.218} C_VEL
LIN {X 0,Y 273.198,Z 865.321,A -85,B 0,C 180,E1 -18744.307,E2 -18744.307} C_VEL
LIN {X 0,Y 277.208,Z 856.255,A -85,B 0,C 180,E1 -18746.34,E2 -18746.34} C_VEL
LIN {X 0,Y 280.241,Z 848.574,A -85,B 0,C 180,E1 -18747.79,E2 -18747.79} C_VEL
LIN {X 0,Y 280.388,Z 846.228,A -85,B 0,C 180,E1 -18748.418,E2 -18748.418} C_VEL
LIN {X 0,Y 279.48,Z 843.651,A -85,B 0,C 180,E1 -18749.482,E2 -18749.482} C_VEL
LIN {X 0,Y 276.511,Z 840.91,A -85,B 0,C 180,E1 -18751.396,E2 -18751.396} C_VEL
LIN {X 0,Y 274.251,Z 838.757,A -85,B 0,C 180,E1 -18752.996,E2 -18752.996} C_VEL
LIN {X 0,Y 273.622,Z 837.247,A -85,B 0,C 180,E1 -18753.79,E2 -18753.79} C_VEL
LIN {X 0,Y 272.251,Z 832.562,A -85,B 0,C 180,E1 -18756.424,E2 -18756.424} C_VEL
LIN {X 0,Y 270.941,Z 829.741,A -85,B 0,C 180,E1 -18758.906,E2 -18758.906} C_VEL
LIN {X 0,Y 270.172,Z 828.334,A -85,B 0,C 180,E1 -18761.029,E2 -18761.029} C_VEL
LIN {X 0,Y 269.898,Z 827.607,A -85,B 0,C 180,E1 -18763.188,E2 -18763.188} C_VEL
LIN {X 0,Y 269.897,Z 828.058,A -85,B 0,C 180,E1 -18765.326,E2 -18765.326} C_VEL
LIN {X 0,Y 270.072,Z 829.796,A -85,B 0,C 180,E1 -18767.422,E2 -18767.422} C_VEL
LIN {X 0,Y 270.972,Z 833.526,A -85,B 0,C 180,E1 -18770.231,E2 -18770.231} C_VEL
LIN {X 0,Y 271.387,Z 836.255,A -85,B 0,C 180,E1 -18771.573,E2 -18771.573} C_VEL
LIN {X 0,Y 271.62,Z 839.923,A -85,B 0,C 180,E1 -18772.943,E2 -18772.943} C_VEL
LIN {X 0,Y 271.218,Z 849.797,A -85,B 0,C 180,E1 -18775.683,E2 -18775.683} C_VEL
LIN {X 0,Y 270.177,Z 860.77,A -85,B 0,C 180,E1 -18778.382,E2 -18778.382} C_VEL
LIN {X 0,Y 268.374,Z 871.313,A -85,B 0,C 180,E1 -18780.845,E2 -18780.845} C_VEL
LIN {X 0,Y 265.753,Z 880.167,A -85,B 0,C 180,E1 -18782.859,E2 -18782.859} C_VEL
LIN {X 0,Y 262.844,Z 887.626,A -85,B 0,C 180,E1 -18784.671,E2 -18784.671} C_VEL
LIN {X 0,Y 258.48,Z 896.728,A -85,B 0,C 180,E1 -18787.204,E2 -18787.204} C_VEL
LIN {X 0,Y 254.474,Z 905.01,A -85,B 0,C 180,E1 -18790.141,E2 -18790.141} C_VEL
LIN {X 0,Y 251.743,Z 911.026,A -85,B 0,C 180,E1 -18792.954,E2 -18792.954} C_VEL
LIN {X 0,Y 249.308,Z 916.182,A -85,B 0,C 180,E1 -18796.136,E2 -18796.136} C_VEL
LIN {X 0,Y 248.161,Z 918.98,A -85,B 0,C 180,E1 -18798.566,E2 -18798.566} C_VEL
LIN {X 0,Y 247.641,Z 920.385,A -85,B 0,C 180,E1 -18800.196,E2 -18800.196} C_VEL
LIN {X 0,Y 247.168,Z 922.01,A -85,B 0,C 180,E1 -18803.469,E2 -18803.469} C_VEL
LIN {X 0,Y 247.17,Z 922.257,A -85,B 0,C 180,E1 -18805.107,E2 -18805.107} C_VEL
LIN {X 0,Y 247.196,Z 922.113,A -85,B 0,C 180,E1 -18806.74,E2 -18806.74} C_VEL
LIN {X 0,Y 247.583,Z 921.279,A -85,B 0,C 180,E1 -18808.983,E2 -18808.983} C_VEL
LIN {X 0,Y 247.605,Z 922.098,A -85,B 0,C 180,E1 -18810,E2 -18810} C_VEL
LIN {X 0,Y 247.255,Z 923.054,A -85,B 0,C 180,E1 -18811.629,E2 -18811.629} C_VEL
LIN {X 0,Y 247.146,Z 923.588,A -85,B 0,C 180,E1 -18813.26,E2 -18813.26} C_VEL
LIN {X 0,Y 247.06,Z 923.687,A -85,B 0,C 180,E1 -18815.347,E2 -18815.347} C_VEL
LIN {X 0,Y 247.278,Z 922.832,A -85,B 0,C 180,E1 -18818.17,E2 -18818.17} C_VEL
LIN {X 0,Y 248.138,Z 920.45,A -85,B 0,C 180,E1 -18821.435,E2 -18821.435} C_VEL
LIN {X 0,Y 249.798,Z 916.506,A -85,B 0,C 180,E1 -18824.668,E2 -18824.668} C_VEL
LIN {X 0,Y 252.476,Z 911.056,A -85,B 0,C 180,E1 -18827.83,E2 -18827.83} C_VEL
LIN {X 0,Y 255.828,Z 903.857,A -85,B 0,C 180,E1 -18830.924,E2 -18830.924} C_VEL
LIN {X 0,Y 259.617,Z 896.074,A -85,B 0,C 180,E1 -18833.534,E2 -18833.534} C_VEL
LIN {X 0,Y 264.26,Z 886.535,A -85,B 0,C 180,E1 -18836.029,E2 -18836.029} C_VEL
LIN {X 0,Y 267.732,Z 877.179,A -85,B 0,C 180,E1 -18838.197,E2 -18838.197} C_VEL
LIN {X 0,Y 269.328,Z 870.675,A -85,B 0,C 180,E1 -18839.722,E2 -18839.722} C_VEL
LIN {X 0,Y 270.404,Z 862.137,A -85,B 0,C 180,E1 -18841.831,E2 -18841.831} C_VEL
LIN {X 0,Y 270.661,Z 853.695,A -85,B 0,C 180,E1 -18844.145,E2 -18844.145} C_VEL
LIN {X 0,Y 270.499,Z 846.681,A -85,B 0,C 180,E1 -18846.346,E2 -18846.346} C_VEL
LIN {X 0,Y 270.196,Z 842.446,A -85,B 0,C 180,E1 -18847.908,E2 -18847.908} C_VEL
LIN {X 0,Y 270.021,Z 839.352,A -85,B 0,C 180,E1 -18849.213,E2 -18849.213} C_VEL
LIN {X 0,Y 269.155,Z 835.424,A -85,B 0,C 180,E1 -18851.769,E2 -18851.769} C_VEL
LIN {X 0,Y 269.045,Z 833.902,A -85,B 0,C 180,E1 -18852.993,E2 -18852.993} C_VEL
LIN {X 0,Y 268.982,Z 832.119,A -85,B 0,C 180,E1 -18855.132,E2 -18855.132} C_VEL
LIN {X 0,Y 269.041,Z 831.705,A -85,B 0,C 180,E1 -18857.219,E2 -18857.219} C_VEL
LIN {X 0,Y 269.369,Z 832.319,A -85,B 0,C 180,E1 -18859.286,E2 -18859.286} C_VEL
LIN {X 0,Y 270.256,Z 833.401,A -85,B 0,C 180,E1 -18861.381,E2 -18861.381} C_VEL
LIN {X 0,Y 271.881,Z 836.329,A -85,B 0,C 180,E1 -18864.205,E2 -18864.205} C_VEL
LIN {X 0,Y 273.256,Z 840.645,A -85,B 0,C 180,E1 -18866.698,E2 -18866.698} C_VEL
LIN {X 0,Y 274.475,Z 846.271,A -85,B 0,C 180,E1 -18869.194,E2 -18869.194} C_VEL
LIN {X 0,Y 275.01,Z 852.316,A -85,B 0,C 180,E1 -18871.405,E2 -18871.405} C_VEL
LIN {X 0,Y 274.737,Z 853.593,A -85,B 0,C 180,E1 -18871.74,E2 -18871.74} C_VEL
LIN {X 0,Y 270.178,Z 863.222,A -85,B 0,C 180,E1 -18873.753,E2 -18873.753} C_VEL
LIN {X 0,Y 265.336,Z 872.443,A -85,B 0,C 180,E1 -18876.174,E2 -18876.174} C_VEL
LIN {X 0,Y 261.102,Z 879.872,A -85,B 0,C 180,E1 -18878.691,E2 -18878.691} C_VEL
LIN {X 0,Y 258.053,Z 884.985,A -85,B 0,C 180,E1 -18880.923,E2 -18880.923} C_VEL
LIN {X 0,Y 254.5,Z 890.356,A -85,B 0,C 180,E1 -18883.968,E2 -18883.968} C_VEL
LIN {X 0,Y 251.725,Z 894.021,A -85,B 0,C 180,E1 -18887.092,E2 -18887.092} C_VEL
LIN {X 0,Y 249.823,Z 896.199,A -85,B 0,C 180,E1 -18890.281,E2 -18890.281} C_VEL
LIN {X 0,Y 248.836,Z 896.741,A -85,B 0,C 180,E1 -18891.88,E2 -18891.88} C_VEL
LIN {X 0,Y 247.966,Z 896.621,A -85,B 0,C 180,E1 -18895.121,E2 -18895.121} C_VEL
LIN {X 0,Y 247.639,Z 896.015,A -85,B 0,C 180,E1 -18896.744,E2 -18896.744} C_VEL
LIN {X 0,Y 247.377,Z 895.027,A -85,B 0,C 180,E1 -18898.37,E2 -18898.37} C_VEL
LIN {X 0,Y 247.226,Z 891.802,A -85,B 0,C 180,E1 -18901.627,E2 -18901.627} C_VEL
LIN {X 0,Y 247.316,Z 888.293,A -85,B 0,C 180,E1 -18904.072,E2 -18904.072} C_VEL
LIN {X 0,Y 247.503,Z 883.704,A -85,B 0,C 180,E1 -18906.52,E2 -18906.52} C_VEL
LIN {X 0,Y 248.049,Z 876.884,A -85,B 0,C 180,E1 -18909.374,E2 -18909.374} C_VEL
LIN {X 0,Y 248.855,Z 869.531,A -85,B 0,C 180,E1 -18911.813,E2 -18911.813} C_VEL
LIN {X 0,Y 249.914,Z 860.558,A -85,B 0,C 180,E1 -18914.243,E2 -18914.243} C_VEL
LIN {X 0,Y 251.236,Z 850.549,A -85,B 0,C 180,E1 -18916.451,E2 -18916.451} C_VEL
LIN {X 0,Y 252.57,Z 839.957,A -85,B 0,C 180,E1 -18918.348,E2 -18918.348} C_VEL
LIN {X 0,Y 253.831,Z 828.452,A -85,B 0,C 180,E1 -18920.036,E2 -18920.036} C_VEL
LIN {X 0,Y 254.149,Z 825.303,A -85,B 0,C 180,E1 -18920.432,E2 -18920.432} C_VEL
LIN {X 0,Y 251.97,Z 813.256,A -85,B 0,C 180,E1 -18921.904,E2 -18921.904} C_VEL
LIN {X 0,Y 249.239,Z 798.889,A -85,B 0,C 180,E1 -18923.304,E2 -18923.304} C_VEL
LIN {X 0,Y 247.708,Z 790.635,A -85,B 0,C 180,E1 -18923.955,E2 -18923.955} C_VEL
LIN {X 0,Y 248.232,Z 790.562,A -85,B 0,C 180,E1 -18928.769,E2 -18928.769} C_VEL
LIN {X 0,Y 248.593,Z 790.519,A -85,B 0,C 180,E1 -18932.488,E2 -18932.488} C_VEL
LIN {X 0,Y 248.907,Z 790.481,A -85,B 0,C 180,E1 -18936.364,E2 -18936.364} C_VEL
LIN {X 0,Y 248.984,Z 790.469,A -85,B 0,C 180,E1 -18940.48,E2 -18940.48} C_VEL
LIN {X 0,Y 248.997,Z 790.47,A -85,B 0,C 180,E1 -18942.789,E2 -18942.789} C_VEL
LIN {X 0,Y 249.004,Z 790.465,A -85,B 0,C 180,E1 -18947.36,E2 -18947.36} C_VEL
LIN {X 0,Y 249.019,Z 790.463,A -85,B 0,C 180,E1 -18951.618,E2 -18951.618} C_VEL
LIN {X 0,Y 249.037,Z 790.461,A -85,B 0,C 180,E1 -18955.638,E2 -18955.638} C_VEL
LIN {X 0,Y 248.995,Z 790.468,A -85,B 0,C 180,E1 -18959.465,E2 -18959.465} C_VEL
LIN {X 0,Y 249.028,Z 790.466,A -85,B 0,C 180,E1 -18963.157,E2 -18963.157} C_VEL
LIN {X 0,Y 249.046,Z 790.459,A -85,B 0,C 180,E1 -18966.729,E2 -18966.729} C_VEL
LIN {X 0,Y 249.07,Z 790.457,A -85,B 0,C 180,E1 -18970.208,E2 -18970.208} C_VEL
LIN {X 0,Y 249.169,Z 790.448,A -85,B 0,C 180,E1 -18973.617,E2 -18973.617} C_VEL
LIN {X 0,Y 249.203,Z 790.438,A -85,B 0,C 180,E1 -18976.961,E2 -18976.961} C_VEL
LIN {X 0,Y 249.377,Z 790.419,A -85,B 0,C 180,E1 -18980.52,E2 -18980.52} C_VEL
LIN {X 0,Y 249.418,Z 790.416,A -85,B 0,C 180,E1 -18983.528,E2 -18983.528} C_VEL
LIN {X 0,Y 249.647,Z 790.387,A -85,B 0,C 180,E1 -18988.387,E2 -18988.387} C_VEL
LIN {X 0,Y 249.645,Z 790.387,A -85,B 0,C 180,E1 -18991.613,E2 -18991.613} C_VEL
LIN {X 0,Y 249.418,Z 790.416,A -85,B 0,C 180,E1 -18996.472,E2 -18996.472} C_VEL
LIN {X 0,Y 249.324,Z 790.427,A -85,B 0,C 180,E1 -18999.737,E2 -18999.737} C_VEL
LIN {X 0,Y 249.163,Z 790.447,A -85,B 0,C 180,E1 -19004.706,E2 -19004.706} C_VEL
LIN {X 0,Y 249.095,Z 790.456,A -85,B 0,C 180,E1 -19008.081,E2 -19008.081} C_VEL
LIN {X 0,Y 249.072,Z 790.455,A -85,B 0,C 180,E1 -19011.52,E2 -19011.52} C_VEL
LIN {X 0,Y 249.077,Z 790.456,A -85,B 0,C 180,E1 -19015.461,E2 -19015.461} C_VEL
LIN {X 0,Y 249.03,Z 790.464,A -85,B 0,C 180,E1 -19018.975,E2 -19018.975} C_VEL
LIN {X 0,Y 249.02,Z 790.462,A -85,B 0,C 180,E1 -19022.427,E2 -19022.427} C_VEL
LIN {X 0,Y 249.023,Z 790.464,A -85,B 0,C 180,E1 -19026.347,E2 -19026.347} C_VEL
LIN {X 0,Y 249,Z 790.464,A -85,B 0,C 180,E1 -19030.479,E2 -19030.479} C_VEL
LIN {X 0,Y 248.981,Z 790.47,A -85,B 0,C 180,E1 -19034.885,E2 -19034.885} C_VEL
LIN {X 0,Y 249.005,Z 790.468,A -85,B 0,C 180,E1 -19037.363,E2 -19037.363} C_VEL
LIN {X 0,Y 249.003,Z 790.468,A -85,B 0,C 180,E1 -19041.618,E2 -19041.618} C_VEL
LIN {X 0,Y 248.848,Z 790.488,A -85,B 0,C 180,E1 -19045.611,E2 -19045.611} C_VEL
LIN {X 0,Y 248.482,Z 790.53,A -85,B 0,C 180,E1 -19049.398,E2 -19049.398} C_VEL
LIN {X 0,Y 248.055,Z 790.584,A -85,B 0,C 180,E1 -19053.045,E2 -19053.045} C_VEL
LIN {X 0,Y 247.747,Z 790.626,A -85,B 0,C 180,E1 -19056.298,E2 -19056.298} C_VEL
LIN {X 0,Y 250.415,Z 804.747,A -85,B 0,C 180,E1 -19057.475,E2 -19057.475} C_VEL
LIN {X 0,Y 253.004,Z 818.327,A -85,B 0,C 180,E1 -19058.94,E2 -19058.94} C_VEL
LIN {X 0,Y 253.966,Z 824.951,A -85,B 0,C 180,E1 -19059.764,E2 -19059.764} C_VEL
LIN {X 0,Y 252.662,Z 837.134,A -85,B 0,C 180,E1 -19061.458,E2 -19061.458} C_VEL
LIN {X 0,Y 251.328,Z 848.141,A -85,B 0,C 180,E1 -19063.346,E2 -19063.346} C_VEL
LIN {X 0,Y 249.921,Z 859.378,A -85,B 0,C 180,E1 -19065.757,E2 -19065.757} C_VEL
LIN {X 0,Y 248.842,Z 868.496,A -85,B 0,C 180,E1 -19068.186,E2 -19068.186} C_VEL
LIN {X 0,Y 248.03,Z 875.944,A -85,B 0,C 180,E1 -19070.625,E2 -19070.625} C_VEL
LIN {X 0,Y 247.502,Z 882.905,A -85,B 0,C 180,E1 -19073.48,E2 -19073.48} C_VEL
LIN {X 0,Y 247.262,Z 887.561,A -85,B 0,C 180,E1 -19075.927,E2 -19075.927} C_VEL
LIN {X 0,Y 247.201,Z 891.128,A -85,B 0,C 180,E1 -19078.373,E2 -19078.373} C_VEL
LIN {X 0,Y 247.338,Z 894.396,A -85,B 0,C 180,E1 -19081.63,E2 -19081.63} C_VEL
LIN {X 0,Y 247.579,Z 895.428,A -85,B 0,C 180,E1 -19083.256,E2 -19083.256} C_VEL
LIN {X 0,Y 248.212,Z 896.301,A -85,B 0,C 180,E1 -19086.505,E2 -19086.505} C_VEL
LIN {X 0,Y 248.811,Z 896.181,A -85,B 0,C 180,E1 -19088.121,E2 -19088.121} C_VEL
LIN {X 0,Y 250.124,Z 895.283,A -85,B 0,C 180,E1 -19090.443,E2 -19090.443} C_VEL
LIN {X 0,Y 251.623,Z 893.484,A -85,B 0,C 180,E1 -19092.913,E2 -19092.913} C_VEL
LIN {X 0,Y 254.299,Z 889.831,A -85,B 0,C 180,E1 -19096.045,E2 -19096.045} C_VEL
LIN {X 0,Y 257.879,Z 884.432,A -85,B 0,C 180,E1 -19099.091,E2 -19099.091} C_VEL
LIN {X 0,Y 260.91,Z 879.288,A -85,B 0,C 180,E1 -19101.326,E2 -19101.326} C_VEL
LIN {X 0,Y 265.142,Z 871.774,A -85,B 0,C 180,E1 -19103.844,E2 -19103.844} C_VEL
LIN {X 0,Y 269.87,Z 862.564,A -85,B 0,C 180,E1 -19106.279,E2 -19106.279} C_VEL
LIN {X 0,Y 275.021,Z 851.158,A -85,B 0,C 180,E1 -19108.642,E2 -19108.642} C_VEL
LIN {X 0,Y 275.02,Z 846.212,A -85,B 0,C 180,E1 -19110.221,E2 -19110.221} C_VEL
LIN {X 0,Y 274.218,Z 840.057,A -85,B 0,C 180,E1 -19112.564,E2 -19112.564} C_VEL
LIN {X 0,Y 273.622,Z 837.247,A -85,B 0,C 180,E1 -19113.79,E2 -19113.79} C_VEL
LIN {X 0,Y 273.12,Z 835.935,A -85,B 0,C 180,E1 -19114.558,E2 -19114.558} C_VEL
LIN {X 0,Y 272.2,Z 835.201,A -85,B 0,C 180,E1 -19115.349,E2 -19115.349} C_VEL
LIN {X 0,Y 270.054,Z 834.894,A -85,B 0,C 180,E1 -19116.967,E2 -19116.967} C_VEL
LIN {X 0,Y 267.26,Z 835.221,A -85,B 0,C 180,E1 -19119.499,E2 -19119.499} C_VEL
LIN {X 0,Y 266.849,Z 834.943,A -85,B 0,C 180,E1 -19120.362,E2 -19120.362} C_VEL
LIN {X 0,Y 266.52,Z 833.85,A -85,B 0,C 180,E1 -19123.285,E2 -19123.285} C_VEL
LIN {X 0,Y 266.506,Z 834.42,A -85,B 0,C 180,E1 -19125.401,E2 -19125.401} C_VEL
LIN {X 0,Y 266.621,Z 836.323,A -85,B 0,C 180,E1 -19127.569,E2 -19127.569} C_VEL
LIN {X 0,Y 267.161,Z 839.061,A -85,B 0,C 180,E1 -19129.721,E2 -19129.721} C_VEL
LIN {X 0,Y 267.419,Z 842.323,A -85,B 0,C 180,E1 -19131.381,E2 -19131.381} C_VEL
LIN {X 0,Y 267.252,Z 846.307,A -85,B 0,C 180,E1 -19132.783,E2 -19132.783} C_VEL
LIN {X 0,Y 266.286,Z 855.131,A -85,B 0,C 180,E1 -19135.333,E2 -19135.333} C_VEL
LIN {X 0,Y 264.692,Z 865.129,A -85,B 0,C 180,E1 -19137.925,E2 -19137.925} C_VEL
LIN {X 0,Y 262.49,Z 874.662,A -85,B 0,C 180,E1 -19140.309,E2 -19140.309} C_VEL
LIN {X 0,Y 258.642,Z 885.17,A -85,B 0,C 180,E1 -19142.926,E2 -19142.926} C_VEL
LIN {X 0,Y 253.961,Z 894.489,A -85,B 0,C 180,E1 -19145.474,E2 -19145.474} C_VEL
LIN {X 0,Y 250.369,Z 901.226,A -85,B 0,C 180,E1 -19147.732,E2 -19147.732} C_VEL
LIN {X 0,Y 247.38,Z 906.851,A -85,B 0,C 180,E1 -19150.067,E2 -19150.067} C_VEL
LIN {X 0,Y 244.269,Z 912.841,A -85,B 0,C 180,E1 -19153.279,E2 -19153.279} C_VEL
LIN {X 0,Y 241.899,Z 917.286,A -85,B 0,C 180,E1 -19156.56,E2 -19156.56} C_VEL
LIN {X 0,Y 240.628,Z 920.159,A -85,B 0,C 180,E1 -19159.907,E2 -19159.907} C_VEL
LIN {X 0,Y 240.082,Z 921.584,A -85,B 0,C 180,E1 -19163.276,E2 -19163.276} C_VEL
LIN {X 0,Y 240.091,Z 921.724,A -85,B 0,C 180,E1 -19164.962,E2 -19164.962} C_VEL
LIN {X 0,Y 240.446,Z 920.778,A -85,B 0,C 180,E1 -19168.325,E2 -19168.325} C_VEL
LIN {X 0,Y 240.553,Z 920.514,A -85,B 0,C 180,E1 -19169.163,E2 -19169.163} C_VEL
LIN {X 0,Y 240.566,Z 921.212,A -85,B 0,C 180,E1 -19170,E2 -19170} C_VEL
LIN {X 0,Y 240.076,Z 922.904,A -85,B 0,C 180,E1 -19173.356,E2 -19173.356} C_VEL
LIN {X 0,Y 239.996,Z 923.164,A -85,B 0,C 180,E1 -19175.333,E2 -19175.333} C_VEL
LIN {X 0,Y 240.223,Z 922.491,A -85,B 0,C 180,E1 -19178.411,E2 -19178.411} C_VEL
LIN {X 0,Y 241.161,Z 920.335,A -85,B 0,C 180,E1 -19181.771,E2 -19181.771} C_VEL
LIN {X 0,Y 242.947,Z 916.732,A -85,B 0,C 180,E1 -19185.091,E2 -19185.091} C_VEL
LIN {X 0,Y 245.742,Z 911.526,A -85,B 0,C 180,E1 -19188.336,E2 -19188.336} C_VEL
LIN {X 0,Y 248.62,Z 905.952,A -85,B 0,C 180,E1 -19191.02,E2 -19191.02} C_VEL
LIN {X 0,Y 252.607,Z 898.544,A -85,B 0,C 180,E1 -19193.792,E2 -19193.792} C_VEL
LIN {X 0,Y 257.334,Z 889.767,A -85,B 0,C 180,E1 -19196.347,E2 -19196.347} C_VEL
LIN {X 0,Y 260.625,Z 882.614,A -85,B 0,C 180,E1 -19198.158,E2 -19198.158} C_VEL
LIN {X 0,Y 262.857,Z 876.479,A -85,B 0,C 180,E1 -19199.646,E2 -19199.646} C_VEL
LIN {X 0,Y 264.658,Z 868.15,A -85,B 0,C 180,E1 -19201.812,E2 -19201.812} C_VEL
LIN {X 0,Y 265.526,Z 861.156,A -85,B 0,C 180,E1 -19203.768,E2 -19203.768} C_VEL
LIN {X 0,Y 265.942,Z 853.229,A -85,B 0,C 180,E1 -19206.283,E2 -19206.283} C_VEL
LIN {X 0,Y 265.95,Z 847.329,A -85,B 0,C 180,E1 -19208.55,E2 -19208.55} C_VEL
LIN {X 0,Y 265.863,Z 844.343,A -85,B 0,C 180,E1 -19209.948,E2 -19209.948} C_VEL
LIN {X 0,Y 265.441,Z 841.199,A -85,B 0,C 180,E1 -19212.152,E2 -19212.152} C_VEL
LIN {X 0,Y 265.375,Z 838.918,A -85,B 0,C 180,E1 -19214.351,E2 -19214.351} C_VEL
LIN {X 0,Y 265.39,Z 838.114,A -85,B 0,C 180,E1 -19215.644,E2 -19215.644} C_VEL
LIN {X 0,Y 265.494,Z 837.978,A -85,B 0,C 180,E1 -19217.834,E2 -19217.834} C_VEL
LIN {X 0,Y 266.193,Z 839.08,A -85,B 0,C 180,E1 -19220.679,E2 -19220.679} C_VEL
LIN {X 0,Y 267.088,Z 840.688,A -85,B 0,C 180,E1 -19222.754,E2 -19222.754} C_VEL
LIN {X 0,Y 268.001,Z 843.168,A -85,B 0,C 180,E1 -19224.764,E2 -19224.764} C_VEL
LIN {X 0,Y 268.818,Z 846.637,A -85,B 0,C 180,E1 -19226.784,E2 -19226.784} C_VEL
LIN {X 0,Y 269.571,Z 852.246,A -85,B 0,C 180,E1 -19229.356,E2 -19229.356} C_VEL
LIN {X 0,Y 269.606,Z 855.89,A -85,B 0,C 180,E1 -19230.777,E2 -19230.777} C_VEL
LIN {X 0,Y 264.265,Z 866.315,A -85,B 0,C 180,E1 -19233.12,E2 -19233.12} C_VEL
LIN {X 0,Y 259.208,Z 874.968,A -85,B 0,C 180,E1 -19235.575,E2 -19235.575} C_VEL
LIN {X 0,Y 254.787,Z 881.959,A -85,B 0,C 180,E1 -19238.136,E2 -19238.136} C_VEL
LIN {X 0,Y 250.586,Z 888.162,A -85,B 0,C 180,E1 -19241.182,E2 -19241.182} C_VEL
LIN {X 0,Y 247.819,Z 891.729,A -85,B 0,C 180,E1 -19243.524,E2 -19243.524} C_VEL
LIN {X 0,Y 244.918,Z 895.138,A -85,B 0,C 180,E1 -19246.727,E2 -19246.727} C_VEL
LIN {X 0,Y 242.88,Z 896.982,A -85,B 0,C 180,E1 -19250,E2 -19250} C_VEL
LIN {X 0,Y 241.866,Z 897.389,A -85,B 0,C 180,E1 -19251.644,E2 -19251.644} C_VEL
LIN {X 0,Y 240.912,Z 897.054,A -85,B 0,C 180,E1 -19254.978,E2 -19254.978} C_VEL
LIN {X 0,Y 240.57,Z 896.308,A -85,B 0,C 180,E1 -19256.649,E2 -19256.649} C_VEL
LIN {X 0,Y 240.165,Z 893.652,A -85,B 0,C 180,E1 -19259.998,E2 -19259.998} C_VEL
LIN {X 0,Y 240.161,Z 890.594,A -85,B 0,C 180,E1 -19262.514,E2 -19262.514} C_VEL
LIN {X 0,Y 240.257,Z 885.826,A -85,B 0,C 180,E1 -19265.427,E2 -19265.427} C_VEL
LIN {X 0,Y 240.758,Z 879.423,A -85,B 0,C 180,E1 -19268.391,E2 -19268.391} C_VEL
LIN {X 0,Y 241.587,Z 871.283,A -85,B 0,C 180,E1 -19271.323,E2 -19271.323} C_VEL
LIN {X 0,Y 242.587,Z 862.558,A -85,B 0,C 180,E1 -19273.826,E2 -19273.826} C_VEL
LIN {X 0,Y 243.989,Z 851.914,A -85,B 0,C 180,E1 -19276.309,E2 -19276.309} C_VEL
LIN {X 0,Y 245.45,Z 840.994,A -85,B 0,C 180,E1 -19278.357,E2 -19278.357} C_VEL
LIN {X 0,Y 246.774,Z 828.964,A -85,B 0,C 180,E1 -19280.199,E2 -19280.199} C_VEL
LIN {X 0,Y 247.079,Z 825.842,A -85,B 0,C 180,E1 -19280.608,E2 -19280.608} C_VEL
LIN {X 0,Y 244.99,Z 814.318,A -85,B 0,C 180,E1 -19282.061,E2 -19282.061} C_VEL
LIN {X 0,Y 242.448,Z 800.938,A -85,B 0,C 180,E1 -19283.422,E2 -19283.422} C_VEL
LIN {X 0,Y 240.699,Z 791.509,A -85,B 0,C 180,E1 -19284.206,E2 -19284.206} C_VEL
LIN {X 0,Y 241.22,Z 791.435,A -85,B 0,C 180,E1 -19289.066,E2 -19289.066} C_VEL
LIN {X 0,Y 241.64,Z 791.382,A -85,B 0,C 180,E1 -19293.544,E2 -19293.544} C_VEL
LIN {X 0,Y 241.824,Z 791.36,A -85,B 0,C 180,E1 -19295.536,E2 -19295.536} C_VEL
LIN {X 0,Y 241.929,Z 791.345,A -85,B 0,C 180,E1 -19299.722,E2 -19299.722} C_VEL
LIN {X 0,Y 241.914,Z 791.349,A -85,B 0,C 180,E1 -19304.203,E2 -19304.203} C_VEL
LIN {X 0,Y 241.928,Z 791.346,A -85,B 0,C 180,E1 -19308.075,E2 -19308.075} C_VEL
LIN {X 0,Y 241.98,Z 791.341,A -85,B 0,C 180,E1 -19312.416,E2 -19312.416} C_VEL
LIN {X 0,Y 241.973,Z 791.341,A -85,B 0,C 180,E1 -19316.506,E2 -19316.506} C_VEL
LIN {X 0,Y 241.97,Z 791.341,A -85,B 0,C 180,E1 -19320.611,E2 -19320.611} C_VEL
LIN {X 0,Y 242.025,Z 791.335,A -85,B 0,C 180,E1 -19324.178,E2 -19324.178} C_VEL
LIN {X 0,Y 242.014,Z 791.334,A -85,B 0,C 180,E1 -19328.315,E2 -19328.315} C_VEL
LIN {X 0,Y 242.107,Z 791.327,A -85,B 0,C 180,E1 -19333.316,E2 -19333.316} C_VEL
LIN {X 0,Y 242.168,Z 791.317,A -85,B 0,C 180,E1 -19338.279,E2 -19338.279} C_VEL
LIN {X 0,Y 242.376,Z 791.295,A -85,B 0,C 180,E1 -19341.664,E2 -19341.664} C_VEL
LIN {X 0,Y 242.391,Z 791.29,A -85,B 0,C 180,E1 -19343.34,E2 -19343.34} C_VEL
LIN {X 0,Y 242.607,Z 791.264,A -85,B 0,C 180,E1 -19348.34,E2 -19348.34} C_VEL
LIN {X 0,Y 242.604,Z 791.264,A -85,B 0,C 180,E1 -19351.66,E2 -19351.66} C_VEL
LIN {X 0,Y 242.39,Z 791.29,A -85,B 0,C 180,E1 -19356.66,E2 -19356.66} C_VEL
LIN {X 0,Y 242.252,Z 791.309,A -85,B 0,C 180,E1 -19360.024,E2 -19360.024} C_VEL
LIN {X 0,Y 242.118,Z 791.322,A -85,B 0,C 180,E1 -19365.144,E2 -19365.144} C_VEL
LIN {X 0,Y 242.034,Z 791.337,A -85,B 0,C 180,E1 -19368.627,E2 -19368.627} C_VEL
LIN {X 0,Y 241.995,Z 791.338,A -85,B 0,C 180,E1 -19372.182,E2 -19372.182} C_VEL
LIN {X 0,Y 242.025,Z 791.335,A -85,B 0,C 180,E1 -19375.822,E2 -19375.822} C_VEL
LIN {X 0,Y 241.962,Z 791.342,A -85,B 0,C 180,E1 -19379.59,E2 -19379.59} C_VEL
LIN {X 0,Y 241.973,Z 791.341,A -85,B 0,C 180,E1 -19383.494,E2 -19383.494} C_VEL
LIN {X 0,Y 241.98,Z 791.341,A -85,B 0,C 180,E1 -19387.584,E2 -19387.584} C_VEL
LIN {X 0,Y 241.928,Z 791.346,A -85,B 0,C 180,E1 -19391.925,E2 -19391.925} C_VEL
LIN {X 0,Y 241.921,Z 791.348,A -85,B 0,C 180,E1 -19396.575,E2 -19396.575} C_VEL
LIN {X 0,Y 241.947,Z 791.342,A -85,B 0,C 180,E1 -19400.282,E2 -19400.282} C_VEL
LIN {X 0,Y 241.876,Z 791.353,A -85,B 0,C 180,E1 -19404.447,E2 -19404.447} C_VEL
LIN {X 0,Y 241.537,Z 791.393,A -85,B 0,C 180,E1 -19408.418,E2 -19408.418} C_VEL
LIN {X 0,Y 241.076,Z 791.454,A -85,B 0,C 180,E1 -19412.199,E2 -19412.199} C_VEL
LIN {X 0,Y 240.704,Z 791.503,A -85,B 0,C 180,E1 -19416.056,E2 -19416.056} C_VEL
LIN {X 0,Y 243.429,Z 805.703,A -85,B 0,C 180,E1 -19417.287,E2 -19417.287} C_VEL
LIN {X 0,Y 246.088,Z 819.842,A -85,B 0,C 180,E1 -19418.868,E2 -19418.868} C_VEL
LIN {X 0,Y 246.901,Z 825.455,A -85,B 0,C 180,E1 -19419.594,E2 -19419.594} C_VEL
LIN {X 0,Y 245.595,Z 837.463,A -85,B 0,C 180,E1 -19421.327,E2 -19421.327} C_VEL
LIN {X 0,Y 244.241,Z 848.481,A -85,B 0,C 180,E1 -19423.279,E2 -19423.279} C_VEL
LIN {X 0,Y 242.783,Z 859.732,A -85,B 0,C 180,E1 -19425.758,E2 -19425.758} C_VEL
LIN {X 0,Y 241.703,Z 868.88,A -85,B 0,C 180,E1 -19428.258,E2 -19428.258} C_VEL
LIN {X 0,Y 240.911,Z 876.355,A -85,B 0,C 180,E1 -19430.769,E2 -19430.769} C_VEL
LIN {X 0,Y 240.451,Z 882.414,A -85,B 0,C 180,E1 -19433.288,E2 -19433.288} C_VEL
LIN {X 0,Y 240.165,Z 887.261,A -85,B 0,C 180,E1 -19435.806,E2 -19435.806} C_VEL
LIN {X 0,Y 240.129,Z 891.031,A -85,B 0,C 180,E1 -19438.325,E2 -19438.325} C_VEL
LIN {X 0,Y 240.128,Z 892.986,A -85,B 0,C 180,E1 -19440.002,E2 -19440.002} C_VEL
LIN {X 0,Y 240.511,Z 895.676,A -85,B 0,C 180,E1 -19443.352,E2 -19443.352} C_VEL
LIN {X 0,Y 240.808,Z 896.457,A -85,B 0,C 180,E1 -19445.025,E2 -19445.025} C_VEL
LIN {X 0,Y 241.816,Z 896.813,A -85,B 0,C 180,E1 -19448.357,E2 -19448.357} C_VEL
LIN {X 0,Y 243.721,Z 895.692,A -85,B 0,C 180,E1 -19451.647,E2 -19451.647} C_VEL
LIN {X 0,Y 244.79,Z 894.582,A -85,B 0,C 180,E1 -19453.28,E2 -19453.28} C_VEL
LIN {X 0,Y 247.61,Z 891.185,A -85,B 0,C 180,E1 -19456.491,E2 -19456.491} C_VEL
LIN {X 0,Y 250.359,Z 887.607,A -85,B 0,C 180,E1 -19458.835,E2 -19458.835} C_VEL
LIN {X 0,Y 253.502,Z 883.041,A -85,B 0,C 180,E1 -19461.127,E2 -19461.127} C_VEL
LIN {X 0,Y 257.663,Z 876.511,A -85,B 0,C 180,E1 -19463.725,E2 -19463.725} C_VEL
LIN {X 0,Y 262.497,Z 868.237,A -85,B 0,C 180,E1 -19466.218,E2 -19466.218} C_VEL
LIN {X 0,Y 267.009,Z 859.781,A -85,B 0,C 180,E1 -19468.282,E2 -19468.282} C_VEL
LIN {X 0,Y 269.583,Z 854.567,A -85,B 0,C 180,E1 -19469.334,E2 -19469.334} C_VEL
LIN {X 0,Y 269.912,Z 851.601,A -85,B 0,C 180,E1 -19470.327,E2 -19470.327} C_VEL
LIN {X 0,Y 269.577,Z 845.663,A -85,B 0,C 180,E1 -19472.694,E2 -19472.694} C_VEL
LIN {X 0,Y 269.099,Z 842.045,A -85,B 0,C 180,E1 -19474.399,E2 -19474.399} C_VEL
LIN {X 0,Y 268.571,Z 839.624,A -85,B 0,C 180,E1 -19475.785,E2 -19475.785} C_VEL
LIN {X 0,Y 267.662,Z 836.743,A -85,B 0,C 180,E1 -19478.028,E2 -19478.028} C_VEL
LIN {X 0,Y 266.849,Z 834.943,A -85,B 0,C 180,E1 -19480.362,E2 -19480.362} C_VEL
LIN {X 0,Y 266.274,Z 834.952,A -85,B 0,C 180,E1 -19481.624,E2 -19481.624} C_VEL
LIN {X 0,Y 265.331,Z 836.031,A -85,B 0,C 180,E1 -19482.868,E2 -19482.868} C_VEL
LIN {X 0,Y 262.992,Z 840.955,A -85,B 0,C 180,E1 -19486.167,E2 -19486.167} C_VEL
LIN {X 0,Y 262.872,Z 841.99,A -85,B 0,C 180,E1 -19487.02,E2 -19487.02} C_VEL
LIN {X 0,Y 263.182,Z 844.49,A -85,B 0,C 180,E1 -19489.207,E2 -19489.207} C_VEL
LIN {X 0,Y 263.266,Z 847.254,A -85,B 0,C 180,E1 -19490.732,E2 -19490.732} C_VEL
LIN {X 0,Y 262.86,Z 850.748,A -85,B 0,C 180,E1 -19492.052,E2 -19492.052} C_VEL
LIN {X 0,Y 261.326,Z 859.487,A -85,B 0,C 180,E1 -19494.73,E2 -19494.73} C_VEL
LIN {X 0,Y 259.023,Z 869.559,A -85,B 0,C 180,E1 -19497.521,E2 -19497.521} C_VEL
LIN {X 0,Y 256.747,Z 877.24,A -85,B 0,C 180,E1 -19499.575,E2 -19499.575} C_VEL
LIN {X 0,Y 252.56,Z 887.163,A -85,B 0,C 180,E1 -19502.218,E2 -19502.218} C_VEL
LIN {X 0,Y 246.983,Z 897.092,A -85,B 0,C 180,E1 -19505.183,E2 -19505.183} C_VEL
LIN {X 0,Y 242.788,Z 904.136,A -85,B 0,C 180,E1 -19507.894,E2 -19507.894} C_VEL
LIN {X 0,Y 239.881,Z 909.138,A -85,B 0,C 180,E1 -19510.31,E2 -19510.31} C_VEL
LIN {X 0,Y 236.789,Z 914.379,A -85,B 0,C 180,E1 -19513.622,E2 -19513.622} C_VEL
LIN {X 0,Y 234.967,Z 917.304,A -85,B 0,C 180,E1 -19516.156,E2 -19516.156} C_VEL
LIN {X 0,Y 233.602,Z 919.954,A -85,B 0,C 180,E1 -19519.6,E2 -19519.6} C_VEL
LIN {X 0,Y 233.028,Z 921.096,A -85,B 0,C 180,E1 -19523.071,E2 -19523.071} C_VEL
LIN {X 0,Y 233.042,Z 921.101,A -85,B 0,C 180,E1 -19524.809,E2 -19524.809} C_VEL
LIN {X 0,Y 233.392,Z 919.984,A -85,B 0,C 180,E1 -19528.274,E2 -19528.274} C_VEL
LIN {X 0,Y 233.542,Z 919.518,A -85,B 0,C 180,E1 -19529.138,E2 -19529.138} C_VEL
LIN {X 0,Y 233.546,Z 920.3,A -85,B 0,C 180,E1 -19530,E2 -19530} C_VEL
LIN {X 0,Y 233.009,Z 922.178,A -85,B 0,C 180,E1 -19533.458,E2 -19533.458} C_VEL
LIN {X 0,Y 232.966,Z 922.516,A -85,B 0,C 180,E1 -19536.931,E2 -19536.931} C_VEL
LIN {X 0,Y 233.59,Z 921.364,A -85,B 0,C 180,E1 -19540.4,E2 -19540.4} C_VEL
LIN {X 0,Y 234.948,Z 918.733,A -85,B 0,C 180,E1 -19543.846,E2 -19543.846} C_VEL
LIN {X 0,Y 237.494,Z 914.66,A -85,B 0,C 180,E1 -19547.213,E2 -19547.213} C_VEL
LIN {X 0,Y 240.769,Z 909.066,A -85,B 0,C 180,E1 -19550.504,E2 -19550.504} C_VEL
LIN {X 0,Y 245,Z 901.869,A -85,B 0,C 180,E1 -19553.678,E2 -19553.678} C_VEL
LIN {X 0,Y 249.647,Z 894.049,A -85,B 0,C 180,E1 -19556.32,E2 -19556.32} C_VEL
LIN {X 0,Y 254.044,Z 886.159,A -85,B 0,C 180,E1 -19558.504,E2 -19558.504} C_VEL
LIN {X 0,Y 257.123,Z 878.989,A -85,B 0,C 180,E1 -19560.376,E2 -19560.376} C_VEL
LIN {X 0,Y 258.973,Z 872.252,A -85,B 0,C 180,E1 -19562.244,E2 -19562.244} C_VEL
LIN {X 0,Y 260.416,Z 864.648,A -85,B 0,C 180,E1 -19564.523,E2 -19564.523} C_VEL
LIN {X 0,Y 261.208,Z 857.267,A -85,B 0,C 180,E1 -19567.049,E2 -19567.049} C_VEL
LIN {X 0,Y 261.566,Z 851.81,A -85,B 0,C 180,E1 -19569.32,E2 -19569.32} C_VEL
LIN {X 0,Y 261.671,Z 850.162,A -85,B 0,C 180,E1 -19570.136,E2 -19570.136} C_VEL
LIN {X 0,Y 261.489,Z 845.766,A -85,B 0,C 180,E1 -19573.473,E2 -19573.473} C_VEL
LIN {X 0,Y 261.596,Z 844.141,A -85,B 0,C 180,E1 -19575.69,E2 -19575.69} C_VEL
LIN {X 0,Y 261.677,Z 843.962,A -85,B 0,C 180,E1 -19577.82,E2 -19577.82} C_VEL
LIN {X 0,Y 262.308,Z 845.177,A -85,B 0,C 180,E1 -19580.986,E2 -19580.986} C_VEL
LIN {X 0,Y 263.099,Z 847.064,A -85,B 0,C 180,E1 -19583.262,E2 -19583.262} C_VEL
LIN {X 0,Y 263.718,Z 849.399,A -85,B 0,C 180,E1 -19585.081,E2 -19585.081} C_VEL
LIN {X 0,Y 264.152,Z 852.516,A -85,B 0,C 180,E1 -19586.927,E2 -19586.927} C_VEL
LIN {X 0,Y 264.343,Z 857.615,A -85,B 0,C 180,E1 -19589.358,E2 -19589.358} C_VEL
LIN {X 0,Y 264.109,Z 859.53,A -85,B 0,C 180,E1 -19590.093,E2 -19590.093} C_VEL
LIN {X 0,Y 258.396,Z 869.341,A -85,B 0,C 180,E1 -19592.458,E2 -19592.458} C_VEL
LIN {X 0,Y 253.813,Z 876.439,A -85,B 0,C 180,E1 -19594.582,E2 -19594.582} C_VEL
LIN {X 0,Y 249.707,Z 882.333,A -85,B 0,C 180,E1 -19596.793,E2 -19596.793} C_VEL
LIN {X 0,Y 246.202,Z 887.141,A -85,B 0,C 180,E1 -19599.093,E2 -19599.093} C_VEL
LIN {X 0,Y 242.107,Z 892.132,A -85,B 0,C 180,E1 -19602.252,E2 -19602.252} C_VEL
LIN {X 0,Y 239.575,Z 894.86,A -85,B 0,C 180,E1 -19604.69,E2 -19604.69} C_VEL
LIN {X 0,Y 236.944,Z 897.148,A -85,B 0,C 180,E1 -19608.015,E2 -19608.015} C_VEL
LIN {X 0,Y 235.929,Z 897.766,A -85,B 0,C 180,E1 -19609.702,E2 -19609.702} C_VEL
LIN {X 0,Y 234.901,Z 898.045,A -85,B 0,C 180,E1 -19611.395,E2 -19611.395} C_VEL
LIN {X 0,Y 233.862,Z 897.402,A -85,B 0,C 180,E1 -19614.826,E2 -19614.826} C_VEL
LIN {X 0,Y 233.225,Z 895.284,A -85,B 0,C 180,E1 -19618.271,E2 -19618.271} C_VEL
LIN {X 0,Y 233.058,Z 892.664,A -85,B 0,C 180,E1 -19620.862,E2 -19620.862} C_VEL
LIN {X 0,Y 233.108,Z 889.092,A -85,B 0,C 180,E1 -19623.455,E2 -19623.455} C_VEL
LIN {X 0,Y 233.252,Z 884.338,A -85,B 0,C 180,E1 -19626.115,E2 -19626.115} C_VEL
LIN {X 0,Y 233.8,Z 877.614,A -85,B 0,C 180,E1 -19629.078,E2 -19629.078} C_VEL
LIN {X 0,Y 234.757,Z 868.897,A -85,B 0,C 180,E1 -19632.095,E2 -19632.095} C_VEL
LIN {X 0,Y 235.869,Z 859.619,A -85,B 0,C 180,E1 -19634.669,E2 -19634.669} C_VEL
LIN {X 0,Y 237.237,Z 849.174,A -85,B 0,C 180,E1 -19637.008,E2 -19637.008} C_VEL
LIN {X 0,Y 238.575,Z 838.871,A -85,B 0,C 180,E1 -19638.905,E2 -19638.905} C_VEL
LIN {X 0,Y 239.982,Z 826.144,A -85,B 0,C 180,E1 -19640.797,E2 -19640.797} C_VEL
LIN {X 0,Y 237.648,Z 813.459,A -85,B 0,C 180,E1 -19642.429,E2 -19642.429} C_VEL
LIN {X 0,Y 234.918,Z 799.085,A -85,B 0,C 180,E1 -19643.907,E2 -19643.907} C_VEL
LIN {X 0,Y 233.69,Z 792.38,A -85,B 0,C 180,E1 -19644.493,E2 -19644.493} C_VEL
LIN {X 0,Y 234.203,Z 792.308,A -85,B 0,C 180,E1 -19649.513,E2 -19649.513} C_VEL
LIN {X 0,Y 234.531,Z 792.268,A -85,B 0,C 180,E1 -19652.959,E2 -19652.959} C_VEL
LIN {X 0,Y 234.807,Z 792.236,A -85,B 0,C 180,E1 -19656.769,E2 -19656.769} C_VEL
LIN {X 0,Y 234.882,Z 792.224,A -85,B 0,C 180,E1 -19658.926,E2 -19658.926} C_VEL
LIN {X 0,Y 234.874,Z 792.226,A -85,B 0,C 180,E1 -19663.486,E2 -19663.486} C_VEL
LIN {X 0,Y 234.873,Z 792.228,A -85,B 0,C 180,E1 -19666.51,E2 -19666.51} C_VEL
LIN {X 0,Y 234.913,Z 792.223,A -85,B 0,C 180,E1 -19671.077,E2 -19671.077} C_VEL
LIN {X 0,Y 234.92,Z 792.221,A -85,B 0,C 180,E1 -19675.36,E2 -19675.36} C_VEL
LIN {X 0,Y 234.892,Z 792.224,A -85,B 0,C 180,E1 -19679.426,E2 -19679.426} C_VEL
LIN {X 0,Y 234.961,Z 792.215,A -85,B 0,C 180,E1 -19683.806,E2 -19683.806} C_VEL
LIN {X 0,Y 234.961,Z 792.214,A -85,B 0,C 180,E1 -19688.965,E2 -19688.965} C_VEL
LIN {X 0,Y 235.048,Z 792.205,A -85,B 0,C 180,E1 -19693.091,E2 -19693.091} C_VEL
LIN {X 0,Y 235.1,Z 792.199,A -85,B 0,C 180,E1 -19697.921,E2 -19697.921} C_VEL
LIN {X 0,Y 235.31,Z 792.173,A -85,B 0,C 180,E1 -19701.412,E2 -19701.412} C_VEL
LIN {X 0,Y 235.343,Z 792.167,A -85,B 0,C 180,E1 -19703.14,E2 -19703.14} C_VEL
LIN {X 0,Y 235.566,Z 792.141,A -85,B 0,C 180,E1 -19708.29,E2 -19708.29} C_VEL
LIN {X 0,Y 235.563,Z 792.142,A -85,B 0,C 180,E1 -19711.71,E2 -19711.71} C_VEL
LIN {X 0,Y 235.342,Z 792.167,A -85,B 0,C 180,E1 -19716.86,E2 -19716.86} C_VEL
LIN {X 0,Y 235.2,Z 792.188,A -85,B 0,C 180,E1 -19720.328,E2 -19720.328} C_VEL
LIN {X 0,Y 235.066,Z 792.201,A -85,B 0,C 180,E1 -19725.61,E2 -19725.61} C_VEL
LIN {X 0,Y 234.976,Z 792.213,A -85,B 0,C 180,E1 -19729.208,E2 -19729.208} C_VEL
LIN {X 0,Y 234.938,Z 792.218,A -85,B 0,C 180,E1 -19732.885,E2 -19732.885} C_VEL
LIN {X 0,Y 234.938,Z 792.221,A -85,B 0,C 180,E1 -19736.661,E2 -19736.661} C_VEL
LIN {X 0,Y 234.892,Z 792.224,A -85,B 0,C 180,E1 -19740.574,E2 -19740.574} C_VEL
LIN {X 0,Y 234.92,Z 792.221,A -85,B 0,C 180,E1 -19744.64,E2 -19744.64} C_VEL
LIN {X 0,Y 234.936,Z 792.221,A -85,B 0,C 180,E1 -19748.946,E2 -19748.946} C_VEL
LIN {X 0,Y 234.873,Z 792.228,A -85,B 0,C 180,E1 -19753.49,E2 -19753.49} C_VEL
LIN {X 0,Y 234.874,Z 792.226,A -85,B 0,C 180,E1 -19756.514,E2 -19756.514} C_VEL
LIN {X 0,Y 234.913,Z 792.22,A -85,B 0,C 180,E1 -19761.08,E2 -19761.08} C_VEL
LIN {X 0,Y 234.847,Z 792.231,A -85,B 0,C 180,E1 -19763.901,E2 -19763.901} C_VEL
LIN {X 0,Y 234.614,Z 792.26,A -85,B 0,C 180,E1 -19767.373,E2 -19767.373} C_VEL
LIN {X 0,Y 234.141,Z 792.318,A -85,B 0,C 180,E1 -19771.3,E2 -19771.3} C_VEL
LIN {X 0,Y 233.671,Z 792.414,A -85,B 0,C 180,E1 -19775.811,E2 -19775.811} C_VEL
LIN {X 0,Y 236.249,Z 805.627,A -85,B 0,C 180,E1 -19776.994,E2 -19776.994} C_VEL
LIN {X 0,Y 238.709,Z 819.021,A -85,B 0,C 180,E1 -19778.522,E2 -19778.522} C_VEL
LIN {X 0,Y 239.836,Z 825.752,A -85,B 0,C 180,E1 -19779.414,E2 -19779.414} C_VEL
LIN {X 0,Y 238.49,Z 838.456,A -85,B 0,C 180,E1 -19781.31,E2 -19781.31} C_VEL
LIN {X 0,Y 237.035,Z 849.837,A -85,B 0,C 180,E1 -19783.421,E2 -19783.421} C_VEL
LIN {X 0,Y 235.645,Z 860.086,A -85,B 0,C 180,E1 -19785.758,E2 -19785.758} C_VEL
LIN {X 0,Y 234.564,Z 869.197,A -85,B 0,C 180,E1 -19788.334,E2 -19788.334} C_VEL
LIN {X 0,Y 233.713,Z 877.777,A -85,B 0,C 180,E1 -19791.354,E2 -19791.354} C_VEL
LIN {X 0,Y 233.223,Z 883.644,A -85,B 0,C 180,E1 -19793.952,E2 -19793.952} C_VEL
LIN {X 0,Y 233.071,Z 888.331,A -85,B 0,C 180,E1 -19796.544,E2 -19796.544} C_VEL
LIN {X 0,Y 233.029,Z 891.961,A -85,B 0,C 180,E1 -19799.138,E2 -19799.138} C_VEL
LIN {X 0,Y 233.189,Z 894.625,A -85,B 0,C 180,E1 -19801.729,E2 -19801.729} C_VEL
LIN {X 0,Y 233.764,Z 896.773,A -85,B 0,C 180,E1 -19805.176,E2 -19805.176} C_VEL
LIN {X 0,Y 234.827,Z 897.45,A -85,B 0,C 180,E1 -19808.608,E2 -19808.608} C_VEL
LIN {X 0,Y 236.843,Z 896.565,A -85,B 0,C 180,E1 -19811.99,E2 -19811.99} C_VEL
LIN {X 0,Y 239.394,Z 894.29,A -85,B 0,C 180,E1 -19815.322,E2 -19815.322} C_VEL
LIN {X 0,Y 241.91,Z 891.561,A -85,B 0,C 180,E1 -19817.763,E2 -19817.763} C_VEL
LIN {X 0,Y 246.012,Z 886.529,A -85,B 0,C 180,E1 -19820.924,E2 -19820.924} C_VEL
LIN {X 0,Y 249.498,Z 881.682,A -85,B 0,C 180,E1 -19823.228,E2 -19823.228} C_VEL
LIN {X 0,Y 254.337,Z 874.643,A -85,B 0,C 180,E1 -19825.8,E2 -19825.8} C_VEL
LIN {X 0,Y 259.605,Z 865.98,A -85,B 0,C 180,E1 -19828.28,E2 -19828.28} C_VEL
LIN {X 0,Y 264.53,Z 857.105,A -85,B 0,C 180,E1 -19830.319,E2 -19830.319} C_VEL
LIN {X 0,Y 264.785,Z 852.809,A -85,B 0,C 180,E1 -19832.064,E2 -19832.064} C_VEL
LIN {X 0,Y 264.576,Z 847.561,A -85,B 0,C 180,E1 -19834.567,E2 -19834.567} C_VEL
LIN {X 0,Y 264.338,Z 845.507,A -85,B 0,C 180,E1 -19835.799,E2 -19835.799} C_VEL
LIN {X 0,Y 263.783,Z 842.942,A -85,B 0,C 180,E1 -19837.793,E2 -19837.793} C_VEL
LIN {X 0,Y 263.184,Z 841.255,A -85,B 0,C 180,E1 -19839.86,E2 -19839.86} C_VEL
LIN {X 0,Y 262.889,Z 840.265,A -85,B 0,C 180,E1 -19841.941,E2 -19841.941} C_VEL
LIN {X 0,Y 262.854,Z 840.036,A -85,B 0,C 180,E1 -19844.042,E2 -19844.042} C_VEL
LIN {X 0,Y 262.859,Z 841.154,A -85,B 0,C 180,E1 -19846.213,E2 -19846.213} C_VEL
LIN {X 0,Y 262.872,Z 841.99,A -85,B 0,C 180,E1 -19847.02,E2 -19847.02} C_VEL
LIN {X 0,Y 262.733,Z 843.193,A -85,B 0,C 180,E1 -19847.838,E2 -19847.838} C_VEL
LIN {X 0,Y 261.988,Z 845.945,A -85,B 0,C 180,E1 -19848.976,E2 -19848.976} C_VEL
LIN {X 0,Y 260.818,Z 849.391,A -85,B 0,C 180,E1 -19850.018,E2 -19850.018} C_VEL
LIN {X 0,Y 257.305,Z 859.517,A -85,B 0,C 180,E1 -19852.775,E2 -19852.775} C_VEL
LIN {X 0,Y 255.284,Z 867.197,A -85,B 0,C 180,E1 -19855.163,E2 -19855.163} C_VEL
LIN {X 0,Y 252.596,Z 875.679,A -85,B 0,C 180,E1 -19857.634,E2 -19857.634} C_VEL
LIN {X 0,Y 249.802,Z 882.559,A -85,B 0,C 180,E1 -19859.574,E2 -19859.574} C_VEL
LIN {X 0,Y 245.77,Z 890.359,A -85,B 0,C 180,E1 -19861.847,E2 -19861.847} C_VEL
LIN {X 0,Y 240.662,Z 898.41,A -85,B 0,C 180,E1 -19864.485,E2 -19864.485} C_VEL
LIN {X 0,Y 236.291,Z 905.101,A -85,B 0,C 180,E1 -19867.253,E2 -19867.253} C_VEL
LIN {X 0,Y 232.319,Z 911.111,A -85,B 0,C 180,E1 -19870.563,E2 -19870.563} C_VEL
